C07260=1101.368,312.708,418.200,179.200,17.140,151.820
C07261=1101.362,312.461,418.231,179.196,17.137,151.821
C07262=1101.356,312.212,418.263,179.193,17.135,151.821
C07263=1101.350,311.965,418.294,179.189,17.133,151.821
C07264=1101.345,311.716,418.325,179.186,17.131,151.821
C07265=1101.339,311.469,418.356,179.183,17.129,151.821
C07266=1101.333,311.221,418.387,179.179,17.128,151.822
C07267=1101.327,310.972,418.419,179.175,17.126,151.822
C07268=1101.322,310.725,418.450,179.172,17.124,151.822
C07269=1101.316,310.477,418.481,179.169,17.121,151.822
C07270=1101.310,310.229,418.512,179.165,17.119,151.822
C07271=1101.304,309.981,418.544,179.162,17.117,151.823
C07272=1101.299,309.733,418.575,179.158,17.115,151.823
C07273=1101.293,309.485,418.606,179.156,17.114,151.823
C07274=1101.288,309.237,418.637,179.152,17.112,151.823
C07275=1101.282,308.989,418.667,179.149,17.110,151.824
C07276=1101.276,308.741,418.699,179.145,17.108,151.824
C07277=1101.270,308.493,418.730,179.142,17.106,151.824
C07278=1101.265,308.245,418.761,179.138,17.104,151.824
C07279=1101.259,307.998,418.792,179.135,17.102,151.824
C07280=1101.253,307.749,418.823,179.131,17.100,151.825
C07281=1101.247,307.501,418.853,179.128,17.098,151.825
C07282=1101.242,307.254,418.885,179.124,17.096,151.825
C07283=1101.236,307.006,418.915,179.121,17.094,151.825
C07284=1101.230,306.757,418.947,179.118,17.093,151.826
C07285=1101.225,306.509,418.977,179.115,17.091,151.826
C07286=1101.219,306.262,419.009,179.111,17.089,151.826
C07287=1101.213,306.014,419.039,179.108,17.087,151.826
C07288=1101.208,305.766,419.070,179.104,17.085,151.826
C07289=1101.202,305.517,419.101,179.101,17.083,151.827
C07290=1101.197,305.269,419.132,179.097,17.081,151.827
C07291=1101.191,305.022,419.163,179.094,17.079,151.827
C07292=1101.186,304.774,419.194,179.090,17.078,151.827
C07293=1101.180,304.526,419.224,179.087,17.075,151.828
C07294=1101.174,304.277,419.255,179.084,17.074,151.828
C07295=1101.168,304.029,419.286,179.081,17.072,151.828
C07296=1101.162,303.781,419.316,179.077,17.070,151.828
C07297=1101.154,303.400,419.364,179.072,17.068,151.829
C07298=1101.146,303.018,419.411,179.067,17.065,151.829
C07299=1101.137,302.637,419.458,179.061,17.062,151.830
C07300=1101.128,302.254,419.505,179.056,17.059,151.830
C07301=1101.123,302.006,419.536,179.053,17.057,151.830
C07302=1101.117,301.758,419.567,179.049,17.055,151.830
C07303=1101.111,301.511,419.597,179.045,17.053,151.831
C07304=1101.106,301.262,419.627,179.042,17.051,151.831
C07305=1101.100,301.014,419.658,179.039,17.050,151.831
C07306=1101.095,300.766,419.688,179.036,17.048,151.831
C07307=1101.089,300.518,419.719,179.032,17.046,151.832
C07308=1101.084,300.270,419.749,179.029,17.044,151.832
C07309=1101.078,300.022,419.779,179.025,17.042,151.832
C07310=1101.073,299.774,419.810,179.022,17.040,151.832
C07311=1101.067,299.527,419.841,179.019,17.039,151.833
C07312=1101.061,299.278,419.870,179.015,17.037,151.833
C07313=1101.056,299.030,419.901,179.012,17.035,151.833
C07314=1101.051,298.782,419.932,179.008,17.034,151.834
C07315=1101.045,298.534,419.962,179.005,17.032,151.834
C07316=1101.039,298.286,419.992,179.001,17.030,151.834
C07317=1101.034,298.038,420.023,178.998,17.028,151.834
C07318=1101.028,297.790,420.053,178.995,17.027,151.835
C07319=1101.022,297.542,420.083,178.991,17.025,151.835
C07320=1101.017,297.294,420.114,178.988,17.023,151.835
C07321=1101.011,297.046,420.143,178.984,17.021,151.835
C07322=1101.005,296.798,420.174,178.981,17.019,151.836
C07323=1101.000,296.550,420.204,178.978,17.018,151.836
C07324=1100.994,296.302,420.234,178.974,17.016,151.836
C07325=1100.986,295.953,420.277,178.969,17.014,151.837
C07326=1100.978,295.604,420.319,178.964,17.012,151.837
C07327=1100.970,295.257,420.361,178.960,17.010,151.838
C07328=1100.961,294.908,420.404,178.954,17.007,151.838
C07329=1100.956,294.659,420.433,178.952,17.006,151.838
C07330=1100.950,294.412,420.464,178.948,17.004,151.839
C07331=1100.945,294.164,420.493,178.944,17.002,151.839
C07332=1100.939,293.916,420.523,178.941,17.000,151.839
C07333=1100.934,293.668,420.553,178.938,16.999,151.840
C07334=1100.928,293.420,420.583,178.934,16.997,151.840
C07335=1100.922,293.171,420.613,178.931,16.996,151.840
C07336=1100.917,292.924,420.643,178.927,16.994,151.841
C07337=1100.911,292.675,420.673,178.924,16.992,151.841
C07338=1100.905,292.427,420.703,178.921,16.991,151.841
C07339=1100.900,292.179,420.733,178.917,16.989,151.841
C07340=1100.894,291.931,420.763,178.914,16.987,151.842
C07341=1100.888,291.683,420.793,178.910,16.986,151.842
C07342=1100.883,291.434,420.822,178.907,16.985,151.842
C07343=1100.877,291.186,420.853,178.903,16.983,151.843
C07344=1100.872,290.938,420.882,178.900,16.981,151.843
C07345=1100.866,290.689,420.912,178.896,16.979,151.843
C07346=1100.860,290.442,420.942,178.893,16.978,151.844
C07347=1100.855,290.194,420.971,178.889,16.977,151.844
C07348=1100.849,289.946,421.001,178.886,16.975,151.844
C07349=1100.843,289.678,421.033,178.882,16.973,151.845
C07350=1100.837,289.410,421.065,178.879,16.972,151.845
C07351=1100.830,289.143,421.097,178.875,16.970,151.845
C07352=1100.824,288.875,421.129,178.871,16.968,151.846
C07353=1100.819,288.627,421.159,178.867,16.967,151.846
C07354=1100.814,288.379,421.188,178.864,16.965,151.846
C07355=1100.807,288.132,421.218,178.861,16.964,151.847
C07356=1100.802,287.883,421.248,178.857,16.963,151.847
C07357=1100.796,287.635,421.277,178.853,16.961,151.847
C07358=1100.790,287.387,421.306,178.851,16.960,151.848
C07359=1100.784,287.138,421.336,178.847,16.958,151.848
C07360=1100.779,286.890,421.366,178.843,16.957,151.849
C07361=1100.773,286.642,421.396,178.840,16.955,151.849
C07362=1100.767,286.394,421.425,178.837,16.954,151.849
C07363=1100.762,286.146,421.454,178.833,16.952,151.849
C07364=1100.756,285.898,421.484,178.829,16.950,151.850
C07365=1100.750,285.649,421.513,178.826,16.949,151.850
C07366=1100.745,285.401,421.543,178.823,16.948,151.851
C07367=1100.740,285.153,421.572,178.819,16.946,151.851
C07368=1100.733,284.905,421.601,178.815,16.945,151.851
C07369=1100.728,284.657,421.630,178.812,16.944,151.852
C07370=1100.722,284.408,421.660,178.809,16.942,151.852
C07371=1100.716,284.160,421.689,178.805,16.940,151.852
C07372=1100.711,283.912,421.718,178.801,16.939,151.853
C07373=1100.706,283.664,421.748,178.798,16.938,151.853
C07374=1100.699,283.416,421.777,178.795,16.936,151.853
C07375=1100.694,283.167,421.807,178.791,16.934,151.854
C07376=1100.688,282.920,421.835,178.788,16.933,151.854
C07377=1100.683,282.671,421.865,178.785,16.931,151.854
C07378=1100.678,282.422,421.894,178.781,16.930,151.855
C07379=1100.671,282.174,421.923,178.778,16.929,151.855
C07380=1100.666,281.927,421.952,178.774,16.927,151.856
C07381=1100.660,281.678,421.981,178.771,16.926,151.856
C07382=1100.655,281.430,422.011,178.768,16.925,151.856
C07383=1100.649,281.182,422.041,178.764,16.923,151.857
C07384=1100.644,280.933,422.069,178.760,16.921,151.857
C07385=1100.638,280.685,422.098,178.756,16.920,151.857
C07386=1100.632,280.437,422.127,178.754,16.919,151.858
C07387=1100.626,280.189,422.156,178.750,16.917,151.858
C07388=1100.621,279.941,422.185,178.746,16.916,151.859
C07389=1100.615,279.692,422.214,178.743,16.915,151.859
C07390=1100.609,279.444,422.243,178.739,16.913,151.859
C07391=1100.604,279.196,422.272,178.735,16.912,151.860
C07392=1100.599,278.947,422.301,178.733,16.911,151.860
C07393=1100.592,278.699,422.330,178.729,16.909,151.860
C07394=1100.587,278.452,422.359,178.725,16.908,151.861
C07395=1100.582,278.203,422.388,178.722,16.907,151.861
C07396=1100.575,277.955,422.417,178.718,16.905,151.862
C07397=1100.570,277.707,422.446,178.715,16.903,151.862
C07398=1100.564,277.458,422.474,178.712,16.902,151.862
C07399=1100.558,277.210,422.503,178.708,16.901,151.863
C07400=1100.554,276.962,422.532,178.704,16.900,151.863
C07401=1100.545,276.603,422.574,178.699,16.898,151.864
C07402=1100.537,276.244,422.616,178.695,16.896,151.864
C07403=1100.528,275.886,422.656,178.690,16.894,151.865
C07404=1100.520,275.528,422.698,178.684,16.892,151.865
C07405=1100.515,275.279,422.727,178.681,16.891,151.866
C07406=1100.509,275.031,422.756,178.677,16.890,151.866
C07407=1100.504,274.783,422.784,178.674,16.889,151.867
C07408=1100.498,274.534,422.813,178.671,16.887,151.867
C07409=1100.493,274.287,422.842,178.667,16.886,151.867
C07410=1100.487,274.038,422.870,178.664,16.885,151.868
C07411=1100.481,273.790,422.899,178.660,16.883,151.868
C07412=1100.475,273.542,422.927,178.656,16.882,151.869
C07413=1100.470,273.293,422.956,178.653,16.881,151.869
C07414=1100.464,273.045,422.985,178.650,16.879,151.869
C07415=1100.458,272.796,423.013,178.646,16.878,151.870
C07416=1100.452,272.548,423.042,178.643,16.877,151.870
C07417=1100.447,272.300,423.070,178.639,16.875,151.871
C07418=1100.441,272.052,423.098,178.636,16.875,151.871
C07419=1100.436,271.804,423.128,178.632,16.873,151.871
C07420=1100.430,271.555,423.156,178.628,16.872,151.872
C07421=1100.425,271.307,423.184,178.625,16.871,151.872
C07422=1100.419,271.058,423.212,178.622,16.869,151.873
C07423=1100.412,270.810,423.241,178.619,16.868,151.873
C07424=1100.407,270.562,423.269,178.615,16.867,151.874
C07425=1100.401,270.313,423.298,178.611,16.865,151.874
C07426=1100.397,270.065,423.326,178.608,16.864,151.874
C07427=1100.391,269.816,423.355,178.604,16.863,151.875
C07428=1100.385,269.569,423.383,178.601,16.862,151.875
C07429=1100.379,269.320,423.412,178.598,16.861,151.876
C07430=1100.374,269.072,423.439,178.594,16.860,151.876
C07431=1100.368,268.823,423.468,178.591,16.859,151.876
C07432=1100.362,268.575,423.496,178.587,16.857,151.877
C07433=1100.356,268.326,423.524,178.584,16.856,151.877
C07434=1100.351,268.078,423.552,178.580,16.855,151.878
C07435=1100.345,267.830,423.580,178.576,16.853,151.878
C07436=1100.340,267.582,423.609,178.573,16.853,151.879
C07437=1100.334,267.333,423.637,178.569,16.851,151.879
C07438=1100.328,267.085,423.665,178.566,16.850,151.879
C07439=1100.322,266.837,423.694,178.562,16.849,151.880
C07440=1100.317,266.589,423.722,178.559,16.847,151.880
C07441=1100.312,266.341,423.750,178.556,16.846,151.881
C07442=1100.306,266.092,423.778,178.552,16.845,151.881
C07443=1100.300,265.844,423.806,178.549,16.844,151.882
C07444=1100.294,265.595,423.834,178.545,16.843,151.882
C07445=1100.289,265.347,423.862,178.542,16.842,151.882
C07446=1100.283,265.098,423.890,178.538,16.840,151.883
C07447=1100.277,264.850,423.917,178.534,16.839,151.883
C07448=1100.272,264.602,423.945,178.531,16.838,151.884
C07449=1100.266,264.353,423.973,178.528,16.837,151.884
C07450=1100.261,264.105,424.001,178.524,16.836,151.885
C07451=1100.255,263.856,424.030,178.521,16.835,151.885
C07452=1100.249,263.608,424.058,178.517,16.834,151.886
C07453=1100.240,263.253,424.097,178.513,16.832,151.886
C07454=1100.232,262.897,424.137,178.507,16.830,151.887
C07455=1100.224,262.540,424.177,178.502,16.829,151.888
C07456=1100.216,262.185,424.216,178.497,16.827,151.888
C07457=1100.210,261.936,424.245,178.494,16.827,151.889
C07458=1100.205,261.688,424.273,178.490,16.825,151.889
C07459=1100.198,261.439,424.300,178.487,16.825,151.890
C07460=1100.193,261.191,424.328,178.483,16.823,151.890
C07461=1100.188,260.943,424.356,178.480,16.822,151.890
C07462=1100.181,260.695,424.383,178.476,16.821,151.891
C07463=1100.176,260.446,424.411,178.473,16.820,151.891
C07464=1100.171,260.198,424.439,178.469,16.819,151.892
C07465=1100.164,259.950,424.466,178.465,16.818,151.892
C07466=1100.159,259.701,424.494,178.462,16.817,151.893
C07467=1100.153,259.452,424.522,178.458,16.815,151.893
C07468=1100.147,259.205,424.549,178.455,16.815,151.894
C07469=1100.142,258.956,424.576,178.451,16.813,151.894
C07470=1100.136,258.707,424.605,178.448,16.813,151.895
C07471=1100.130,258.459,424.631,178.444,16.811,151.895
C07472=1100.125,258.211,424.659,178.441,16.811,151.896
C07473=1100.118,257.962,424.687,178.437,16.809,151.896
C07474=1100.113,257.714,424.714,178.434,16.809,151.896
C07475=1100.108,257.466,424.742,178.430,16.807,151.897
C07476=1100.102,257.217,424.769,178.427,16.806,151.897
C07477=1100.096,256.968,424.797,178.423,16.805,151.898
C07478=1100.090,256.720,424.824,178.420,16.804,151.898
C07479=1100.085,256.472,424.852,178.416,16.803,151.899
C07480=1100.079,256.223,424.880,178.413,16.802,151.899
C07481=1100.073,255.975,424.907,178.409,16.801,151.900
C07482=1100.068,255.726,424.934,178.406,16.800,151.900
C07483=1100.062,255.478,424.961,178.402,16.799,151.901
C07484=1100.056,255.229,424.989,178.399,16.798,151.901
C07485=1100.051,254.981,425.016,178.395,16.797,151.902
C07486=1100.045,254.733,425.044,178.392,16.796,151.902
C07487=1100.039,254.484,425.070,178.388,16.795,151.902
C07488=1100.034,254.235,425.098,178.385,16.794,151.903
C07489=1100.028,253.987,425.125,178.381,16.793,151.903
C07490=1100.023,253.739,425.153,178.378,16.792,151.904
C07491=1100.017,253.490,425.179,178.375,16.791,151.904
C07492=1100.012,253.242,425.207,178.371,16.790,151.905
C07493=1100.006,252.994,425.234,178.368,16.788,151.905
C07494=1100.000,252.744,425.261,178.364,16.788,151.906
C07495=1099.994,252.496,425.288,178.360,16.787,151.906
C07496=1099.989,252.248,425.316,178.357,16.786,151.907
C07497=1099.983,252.000,425.343,178.353,16.785,151.907
C07498=1099.978,251.751,425.370,178.350,16.784,151.908
C07499=1099.973,251.503,425.397,178.346,16.783,151.908
C07500=1099.967,251.253,425.424,178.344,16.782,151.908
C07501=1099.961,251.005,425.452,178.340,16.780,151.909
C07502=1099.956,250.757,425.479,178.337,16.779,151.909
C07503=1099.950,250.508,425.505,178.333,16.778,151.910
C07504=1099.945,250.260,425.533,178.329,16.778,151.910
C07505=1099.937,249.901,425.571,178.325,16.776,151.911
C07506=1099.929,249.543,425.611,178.319,16.775,151.912
C07507=1099.921,249.184,425.649,178.314,16.773,151.913
C07508=1099.913,248.825,425.688,178.310,16.772,151.913
C07509=1099.907,248.577,425.715,178.306,16.771,151.914
C07510=1099.902,248.329,425.742,178.303,16.770,151.914
C07511=1099.896,248.079,425.769,178.299,16.768,151.915
C07512=1099.890,247.831,425.796,178.295,16.768,151.915
C07513=1099.885,247.583,425.822,178.292,16.766,151.915
C07514=1099.879,247.334,425.850,178.288,16.766,151.916
C07515=1099.874,247.086,425.876,178.285,16.764,151.916
C07516=1099.868,246.837,425.903,178.282,16.764,151.917
C07517=1099.862,246.589,425.930,178.278,16.763,151.917
C07518=1099.857,246.340,425.957,178.275,16.762,151.918
C07519=1099.851,246.092,425.984,178.271,16.761,151.918
C07520=1099.846,245.843,426.010,178.267,16.760,151.919
C07521=1099.840,245.595,426.037,178.264,16.759,151.919
C07522=1099.835,245.346,426.064,178.260,16.758,151.920
C07523=1099.829,245.098,426.091,178.257,16.757,151.920
C07524=1099.823,244.850,426.117,178.253,16.756,151.921
C07525=1099.818,244.601,426.143,178.250,16.755,151.921
C07526=1099.812,244.352,426.170,178.246,16.754,151.922
C07527=1099.807,244.104,426.197,178.243,16.753,151.922
C07528=1099.801,243.855,426.224,178.240,16.753,151.923
C07529=1099.795,243.607,426.250,178.236,16.752,151.923
C07530=1099.790,243.358,426.276,178.233,16.751,151.924
C07531=1099.784,243.110,426.303,178.229,16.750,151.924
C07532=1099.778,242.861,426.330,178.226,16.749,151.925
C07533=1099.773,242.613,426.356,178.222,16.747,151.925
C07534=1099.767,242.364,426.382,178.219,16.747,151.926
C07535=1099.761,242.116,426.409,178.216,16.746,151.926
C07536=1099.756,241.867,426.436,178.212,16.745,151.927
C07537=1099.750,241.619,426.462,178.208,16.745,151.927
C07538=1099.744,241.370,426.488,178.205,16.743,151.928
C07539=1099.739,241.122,426.515,178.201,16.743,151.928
C07540=1099.733,240.873,426.541,178.198,16.742,151.929
C07541=1099.727,240.624,426.567,178.194,16.741,151.929
C07542=1099.722,240.376,426.594,178.191,16.740,151.930
C07543=1099.716,240.127,426.620,178.187,16.739,151.930
C07544=1099.710,239.878,426.647,178.184,16.738,151.931
C07545=1099.705,239.630,426.673,178.180,16.737,151.931
C07546=1099.699,239.381,426.699,178.177,16.736,151.932
C07547=1099.693,239.133,426.726,178.174,16.736,151.932
C07548=1099.688,238.884,426.752,178.170,16.735,151.933
C07549=1099.682,238.635,426.778,178.167,16.734,151.933
C07550=1099.677,238.386,426.804,178.163,16.733,151.934
C07551=1099.671,238.138,426.831,178.160,16.732,151.934
C07552=1099.665,237.889,426.857,178.156,16.732,151.935
C07553=1099.660,237.641,426.884,178.152,16.731,151.935
C07554=1099.654,237.392,426.910,178.149,16.730,151.936
C07555=1099.649,237.144,426.936,178.145,16.728,151.936
C07556=1099.643,236.895,426.961,178.142,16.728,151.937
C07557=1099.634,236.529,427.001,178.137,16.727,151.938
C07558=1099.626,236.164,427.039,178.132,16.725,151.938
C07559=1099.618,235.798,427.077,178.127,16.724,151.939
C07560=1099.610,235.433,427.115,178.122,16.723,151.940
C07561=1099.604,235.184,427.141,178.119,16.722,151.940
C07562=1099.598,234.936,427.168,178.115,16.721,151.941
C07563=1099.593,234.688,427.193,178.111,16.721,151.941
C07564=1099.587,234.439,427.219,178.108,16.720,151.942
C07565=1099.582,234.191,427.246,178.104,16.719,151.942
C07566=1099.576,233.942,427.271,178.101,16.718,151.943
C07567=1099.571,233.693,427.297,178.098,16.718,151.943
C07568=1099.564,233.444,427.323,178.094,16.716,151.944
C07569=1099.559,233.196,427.349,178.091,16.716,151.944
C07570=1099.554,232.947,427.375,178.087,16.714,151.945
C07571=1099.548,232.698,427.401,178.084,16.714,151.945
C07572=1099.542,232.450,427.426,178.081,16.713,151.946
C07573=1099.536,232.201,427.453,178.077,16.712,151.946
C07574=1099.532,231.953,427.478,178.074,16.711,151.947
C07575=1099.525,231.704,427.504,178.070,16.711,151.948
C07576=1099.520,231.455,427.530,178.066,16.710,151.948
C07577=1099.514,231.206,427.556,178.063,16.709,151.949
C07578=1099.509,230.959,427.582,178.060,16.708,151.949
C07579=1099.503,230.710,427.607,178.056,16.707,151.950
C07580=1099.498,230.461,427.633,178.053,16.707,151.950
C07581=1099.491,230.212,427.659,178.050,16.706,151.951
C07582=1099.486,229.963,427.684,178.046,16.705,151.951
C07583=1099.481,229.715,427.710,178.042,16.705,151.952
C07584=1099.475,229.467,427.735,178.039,16.704,151.952
C07585=1099.469,229.218,427.761,178.035,16.703,151.953
C07586=1099.463,228.969,427.787,178.032,16.702,151.953
C07587=1099.458,228.721,427.812,178.029,16.702,151.954
C07588=1099.452,228.472,427.838,178.025,16.700,151.954
C07589=1099.447,228.223,427.863,178.022,16.700,151.955
C07590=1099.440,227.974,427.889,178.018,16.699,151.955
C07591=1099.436,227.726,427.914,178.014,16.698,151.956
C07592=1099.429,227.477,427.940,178.011,16.698,151.956
C07593=1099.424,227.228,427.966,178.008,16.697,151.957
C07594=1099.418,226.980,427.991,178.004,16.696,151.957
C07595=1099.413,226.731,428.017,178.001,16.695,151.958
C07596=1099.407,226.483,428.042,177.998,16.695,151.959
C07597=1099.401,226.234,428.068,177.994,16.694,151.959
C07598=1099.395,225.986,428.093,177.991,16.693,151.960
C07599=1099.390,225.737,428.119,177.987,16.693,151.960
C07600=1099.384,225.488,428.144,177.983,16.692,151.961
C07601=1099.379,225.240,428.170,177.980,16.691,151.961
C07602=1099.373,224.991,428.194,177.977,16.690,151.962
C07603=1099.368,224.742,428.220,177.973,16.689,151.962
C07604=1099.362,224.494,428.245,177.970,16.689,151.963
C07605=1099.356,224.245,428.271,177.967,16.688,151.963
C07606=1099.351,223.997,428.296,177.963,16.687,151.964
C07607=1099.346,223.747,428.321,177.960,16.686,151.964
C07608=1099.340,223.498,428.347,177.956,16.686,151.965
C07609=1099.331,223.125,428.384,177.951,16.685,151.966
C07610=1099.323,222.751,428.422,177.946,16.683,151.966
C07611=1099.314,222.377,428.460,177.941,16.682,151.967
C07612=1099.306,222.003,428.498,177.936,16.681,151.968
C07613=1099.300,221.754,428.523,177.932,16.680,151.968
C07614=1099.295,221.506,428.548,177.928,16.679,151.969
C07615=1099.289,221.257,428.574,177.925,16.679,151.970
C07616=1099.283,221.008,428.599,177.922,16.678,151.970
C07617=1099.278,220.760,428.624,177.919,16.678,151.971
C07618=1099.272,220.510,428.649,177.915,16.677,151.971
C07619=1099.266,220.261,428.675,177.911,16.676,151.972
C07620=1099.261,220.014,428.700,177.908,16.676,151.972
C07621=1099.255,219.764,428.724,177.904,16.675,151.973
C07622=1099.249,219.516,428.749,177.901,16.674,151.973
C07623=1099.243,219.267,428.774,177.898,16.674,151.974
C07624=1099.238,219.019,428.799,177.895,16.673,151.975
C07625=1099.232,218.770,428.825,177.890,16.672,151.975
C07626=1099.227,218.521,428.849,177.888,16.671,151.976
C07627=1099.221,218.273,428.874,177.884,16.671,151.976
C07628=1099.215,218.023,428.899,177.880,16.670,151.977
C07629=1099.210,217.775,428.924,177.877,16.669,151.977
C07630=1099.204,217.526,428.949,177.874,16.669,151.978
C07631=1099.198,217.278,428.974,177.871,16.668,151.978
C07632=1099.193,217.029,428.999,177.867,16.667,151.979
C07633=1099.187,216.780,429.023,177.863,16.667,151.979
C07634=1099.182,216.531,429.049,177.860,16.666,151.980
C07635=1099.177,216.282,429.073,177.857,16.666,151.980
C07636=1099.170,216.034,429.098,177.853,16.665,151.981
C07637=1099.165,215.785,429.123,177.850,16.664,151.981
C07638=1099.159,215.536,429.147,177.847,16.663,151.982
C07639=1099.153,215.288,429.172,177.843,16.663,151.983
C07640=1099.148,215.039,429.197,177.839,16.662,151.983
C07641=1099.142,214.790,429.221,177.836,16.661,151.984
C07642=1099.137,214.542,429.247,177.833,16.661,151.984
C07643=1099.132,214.293,429.271,177.830,16.660,151.985
C07644=1099.126,214.044,429.296,177.826,16.659,151.985
C07645=1099.120,213.795,429.321,177.822,16.659,151.986
C07646=1099.115,213.547,429.345,177.819,16.658,151.986
C07647=1099.109,213.298,429.369,177.816,16.657,151.987
C07648=1099.103,213.049,429.395,177.812,16.656,151.987
C07649=1099.098,212.801,429.419,177.809,16.656,151.988
C07650=1099.092,212.552,429.444,177.806,16.655,151.988
C07651=1099.087,212.303,429.468,177.802,16.655,151.989
C07652=1099.081,212.054,429.493,177.798,16.654,151.990
C07653=1099.075,211.806,429.518,177.795,16.653,151.990
C07654=1099.070,211.557,429.542,177.792,16.653,151.991
C07655=1099.064,211.308,429.566,177.789,16.652,151.991
C07656=1099.059,211.059,429.591,177.785,16.651,151.992
C07657=1099.053,210.810,429.615,177.781,16.651,151.992
C07658=1099.047,210.562,429.640,177.778,16.650,151.993
C07659=1099.042,210.313,429.664,177.775,16.650,151.993
C07660=1099.035,210.064,429.689,177.772,16.649,151.994
C07661=1099.028,209.694,429.725,177.767,16.648,151.995
C07662=1099.019,209.324,429.761,177.761,16.647,151.995
C07663=1099.010,208.954,429.798,177.756,16.646,151.996
C07664=1099.002,208.584,429.834,177.751,16.645,151.997
C07665=1098.979,207.575,429.932,177.709,16.631,152.003
C07666=1098.974,207.326,429.956,177.705,16.631,152.003
C07667=1098.968,207.078,429.980,177.702,16.632,152.004
C07668=1098.963,206.829,430.003,177.698,16.632,152.005
C07669=1098.957,206.579,430.028,177.694,16.632,152.006
C07670=1098.951,206.331,430.052,177.691,16.632,152.007
C07671=1098.945,206.082,430.076,177.687,16.632,152.007
C07672=1098.940,205.834,430.100,177.683,16.632,152.008
C07673=1098.934,205.585,430.124,177.680,16.632,152.009
C07674=1098.928,205.336,430.147,177.676,16.633,152.010
C07675=1098.923,205.087,430.172,177.673,16.633,152.010
C07676=1098.918,204.839,430.196,177.670,16.633,152.011
C07677=1098.911,204.590,430.220,177.666,16.634,152.012
C07678=1098.906,204.340,430.244,177.662,16.634,152.013
C07679=1098.901,204.092,430.268,177.658,16.634,152.014
C07680=1098.895,203.843,430.291,177.655,16.634,152.014
C07681=1098.890,203.594,430.315,177.651,16.634,152.015
C07682=1098.883,203.345,430.339,177.648,16.635,152.016
C07683=1098.878,203.097,430.363,177.644,16.635,152.017
C07684=1098.873,202.848,430.387,177.640,16.635,152.017
C07685=1098.867,202.599,430.410,177.637,16.635,152.018
C07686=1098.862,202.351,430.435,177.633,16.635,152.019
C07687=1098.855,202.101,430.458,177.630,16.636,152.020
C07688=1098.850,201.852,430.482,177.627,16.636,152.020
C07689=1098.844,201.604,430.506,177.623,16.636,152.021
C07690=1098.838,201.355,430.529,177.619,16.637,152.022
C07691=1098.832,201.106,430.554,177.616,16.637,152.023
C07692=1098.826,200.858,430.577,177.612,16.637,152.024
C07693=1098.821,200.609,430.601,177.608,16.637,152.024
C07694=1098.815,200.360,430.624,177.605,16.637,152.025
C07695=1098.810,200.111,430.648,177.601,16.638,152.026
C07696=1098.804,199.862,430.672,177.598,16.638,152.027
C07697=1098.798,199.613,430.695,177.594,16.639,152.027
C07698=1098.793,199.365,430.719,177.591,16.639,152.028
C07699=1098.787,199.116,430.742,177.587,16.639,152.029
C07700=1098.781,198.867,430.766,177.583,16.639,152.030
C07701=1098.776,198.618,430.789,177.580,16.639,152.030
C07702=1098.769,198.369,430.813,177.576,16.639,152.031
C07703=1098.764,198.120,430.837,177.573,16.639,152.032
C07704=1098.758,197.872,430.861,177.569,16.639,152.033
C07705=1098.752,197.623,430.883,177.566,16.640,152.033
C07706=1098.747,197.374,430.908,177.562,16.641,152.034
C07707=1098.741,197.125,430.931,177.559,16.641,152.035
C07708=1098.736,196.876,430.954,177.555,16.641,152.036
C07709=1098.730,196.628,430.978,177.552,16.641,152.036
C07710=1098.725,196.379,431.001,177.548,16.641,152.037
C07711=1098.718,196.129,431.024,177.544,16.641,152.038
C07712=1098.713,195.881,431.048,177.541,16.641,152.039
C07713=1098.707,195.632,431.071,177.537,16.641,152.039
C07714=1098.701,195.383,431.094,177.534,16.642,152.040
C07715=1098.696,195.134,431.119,177.531,16.642,152.041
C07716=1098.690,194.885,431.141,177.527,16.642,152.042
C07717=1098.685,194.637,431.164,177.524,16.642,152.042
C07718=1098.679,194.388,431.188,177.520,16.643,152.043
C07719=1098.674,194.139,431.212,177.516,16.643,152.044
C07720=1098.668,193.890,431.235,177.513,16.643,152.045
C07721=1098.662,193.641,431.258,177.509,16.643,152.045
C07722=1098.657,193.393,431.282,177.507,16.643,152.046
C07723=1098.651,193.144,431.305,177.503,16.643,152.047
C07724=1098.645,192.895,431.328,177.499,16.644,152.048
C07725=1098.640,192.646,431.351,177.496,16.644,152.048
C07726=1098.633,192.373,431.377,177.492,16.644,152.049
C07727=1098.627,192.099,431.402,177.488,16.644,152.050
C07728=1098.621,191.825,431.428,177.485,16.644,152.051
C07729=1098.615,191.552,431.453,177.480,16.644,152.052
C07730=1098.610,191.303,431.476,177.477,16.645,152.052
C07731=1098.604,191.054,431.499,177.474,16.645,152.053
C07732=1098.599,190.805,431.522,177.470,16.645,152.054
C07733=1098.593,190.557,431.546,177.467,16.645,152.054
C07734=1098.588,190.307,431.569,177.463,16.645,152.055
C07735=1098.582,190.058,431.592,177.460,16.645,152.056
C07736=1098.576,189.810,431.615,177.456,16.645,152.057
C07737=1098.570,189.561,431.638,177.452,16.645,152.058
C07738=1098.565,189.312,431.661,177.450,16.646,152.058
C07739=1098.560,189.063,431.685,177.446,16.646,152.059
C07740=1098.554,188.814,431.708,177.442,16.646,152.060
C07741=1098.548,188.565,431.731,177.439,16.646,152.060
C07742=1098.543,188.316,431.753,177.435,16.646,152.061
C07743=1098.537,188.068,431.776,177.432,16.646,152.062
C07744=1098.532,187.819,431.799,177.428,16.646,152.062
C07745=1098.526,187.570,431.822,177.426,16.646,152.063
C07746=1098.521,187.321,431.845,177.422,16.646,152.064
C07747=1098.515,187.072,431.868,177.418,16.646,152.065
C07748=1098.509,186.823,431.891,177.415,16.647,152.065
C07749=1098.504,186.574,431.914,177.411,16.647,152.066
C07750=1098.498,186.325,431.937,177.408,16.647,152.067
C07751=1098.493,186.076,431.959,177.405,16.647,152.067
C07752=1098.487,185.827,431.982,177.402,16.647,152.068
C07753=1098.482,185.578,432.006,177.398,16.647,152.069
C07754=1098.477,185.329,432.029,177.395,16.647,152.069
C07755=1098.471,185.080,432.052,177.391,16.647,152.070
C07756=1098.465,184.832,432.074,177.388,16.647,152.071
C07757=1098.459,184.583,432.097,177.384,16.647,152.072
C07758=1098.453,184.333,432.119,177.381,16.648,152.072
C07759=1098.448,184.084,432.142,177.378,16.648,152.073
C07760=1098.443,183.836,432.165,177.374,16.648,152.074
C07761=1098.437,183.587,432.188,177.370,16.648,152.075
C07762=1098.430,183.339,432.210,177.367,16.648,152.075
C07763=1098.425,183.090,432.233,177.364,16.649,152.076
C07764=1098.419,182.840,432.255,177.361,16.649,152.077
C07765=1098.413,182.591,432.278,177.357,16.649,152.077
C07766=1098.408,182.343,432.301,177.354,16.649,152.078
C07767=1098.401,182.094,432.323,177.350,16.649,152.079
C07768=1098.396,181.844,432.346,177.346,16.649,152.080
C07769=1098.390,181.596,432.368,177.344,16.649,152.080
C07770=1098.385,181.347,432.391,177.340,16.649,152.081
C07771=1098.379,181.098,432.413,177.337,16.649,152.082
C07772=1098.373,180.849,432.436,177.333,16.650,152.082
C07773=1098.367,180.600,432.459,177.330,16.650,152.083
C07774=1098.362,180.351,432.481,177.327,16.650,152.084
C07775=1098.355,180.102,432.503,177.323,16.650,152.085
C07776=1098.350,179.853,432.526,177.320,16.650,152.085
C07777=1098.345,179.605,432.548,177.316,16.650,152.086
C07778=1098.339,179.356,432.571,177.313,16.650,152.087
C07779=1098.333,179.107,432.593,177.309,16.650,152.087
C07780=1098.327,178.858,432.615,177.306,16.651,152.088
C07781=1098.322,178.609,432.638,177.303,16.651,152.089
C07782=1098.317,178.360,432.660,177.299,16.651,152.090
C07783=1098.310,178.111,432.683,177.296,16.651,152.090
C07784=1098.305,177.862,432.705,177.292,16.651,152.091
C07785=1098.299,177.613,432.728,177.290,16.651,152.092
C07786=1098.293,177.364,432.749,177.286,16.651,152.092
C07787=1098.288,177.115,432.772,177.283,16.651,152.093
C07788=1098.282,176.866,432.794,177.279,16.651,152.094
C07789=1098.276,176.617,432.817,177.276,16.651,152.094
C07790=1098.270,176.343,432.841,177.272,16.651,152.095
C07791=1098.264,176.070,432.865,177.268,16.651,152.096
C07792=1098.258,175.795,432.890,177.265,16.652,152.097
C07793=1098.251,175.521,432.915,177.261,16.652,152.098
C07794=1098.246,175.272,432.937,177.258,16.652,152.098
C07795=1098.240,175.024,432.959,177.254,16.652,152.099
C07796=1098.234,174.774,432.981,177.252,16.652,152.100
C07797=1098.229,174.525,433.004,177.248,16.652,152.100
C07798=1098.224,174.277,433.026,177.244,16.652,152.101
C07799=1098.218,174.027,433.048,177.241,16.652,152.102
C07800=1098.212,173.779,433.070,177.238,16.652,152.102
C07801=1098.206,173.530,433.092,177.235,16.653,152.103
C07802=1098.201,173.281,433.114,177.231,16.653,152.104
C07803=1098.195,173.032,433.137,177.228,16.652,152.104
C07804=1098.190,172.783,433.158,177.225,16.652,152.105
C07805=1098.184,172.534,433.180,177.221,16.652,152.106
C07806=1098.178,172.285,433.203,177.219,16.653,152.106
C07807=1098.173,172.036,433.225,177.215,16.653,152.107
C07808=1098.167,171.787,433.247,177.211,16.653,152.108
C07809=1098.161,171.538,433.269,177.208,16.653,152.108
C07810=1098.156,171.289,433.291,177.205,16.653,152.109
C07811=1098.150,171.040,433.313,177.202,16.653,152.110
C07812=1098.145,170.791,433.335,177.198,16.653,152.110
C07813=1098.139,170.542,433.356,177.195,16.653,152.111
C07814=1098.133,170.293,433.379,177.192,16.653,152.112
C07815=1098.128,170.045,433.400,177.189,16.653,152.112
C07816=1098.122,169.795,433.423,177.186,16.653,152.113
C07817=1098.117,169.546,433.445,177.182,16.653,152.114
C07818=1098.111,169.297,433.466,177.179,16.652,152.114
C07819=1098.106,169.048,433.489,177.175,16.653,152.115
C07820=1098.100,168.800,433.510,177.173,16.653,152.115
C07821=1098.095,168.550,433.533,177.169,16.653,152.116
C07822=1098.089,168.302,433.554,177.166,16.653,152.117
C07823=1098.084,168.052,433.576,177.162,16.652,152.117
C07824=1098.078,167.804,433.597,177.160,16.653,152.118
C07825=1098.073,167.554,433.620,177.156,16.653,152.119
C07826=1098.067,167.306,433.641,177.153,16.653,152.119
C07827=1098.062,167.056,433.663,177.150,16.652,152.120
C07828=1098.055,166.807,433.685,177.146,16.652,152.121
C07829=1098.051,166.558,433.707,177.144,16.653,152.121
C07830=1098.044,166.309,433.728,177.140,16.653,152.122
C07831=1098.040,166.060,433.750,177.137,16.652,152.123
C07832=1098.033,165.811,433.772,177.133,16.652,152.123
C07833=1098.028,165.562,433.793,177.131,16.652,152.124
C07834=1098.022,165.313,433.815,177.127,16.652,152.125
C07835=1098.017,165.064,433.837,177.124,16.652,152.125
C07836=1098.012,164.816,433.858,177.120,16.652,152.126
C07837=1098.006,164.566,433.880,177.117,16.652,152.126
C07838=1098.001,164.318,433.902,177.115,16.652,152.127
C07839=1097.995,164.068,433.924,177.111,16.652,152.128
C07840=1097.990,163.820,433.945,177.108,16.652,152.128
C07841=1097.984,163.570,433.967,177.104,16.652,152.129
C07842=1097.978,163.322,433.988,177.102,16.652,152.130
C07843=1097.973,163.072,434.011,177.099,16.651,152.130
C07844=1097.967,162.824,434.032,177.095,16.651,152.131
C07845=1097.963,162.575,434.054,177.092,16.651,152.131
C07846=1097.957,162.325,434.075,177.088,16.651,152.132
C07847=1097.951,162.077,434.096,177.086,16.651,152.133
C07848=1097.946,161.827,434.118,177.083,16.651,152.133
C07849=1097.940,161.579,434.139,177.079,16.651,152.134
C07850=1097.934,161.329,434.161,177.076,16.651,152.135
C07851=1097.929,161.081,434.183,177.073,16.651,152.135
C07852=1097.923,160.831,434.204,177.070,16.651,152.136
C07853=1097.918,160.582,434.225,177.067,16.650,152.136
C07854=1097.911,160.308,434.249,177.063,16.651,152.137
C07855=1097.905,160.034,434.272,177.059,16.651,152.138
C07856=1097.899,159.759,434.296,177.056,16.651,152.139
C07857=1097.892,159.485,434.320,177.052,16.651,152.139
C07858=1097.887,159.236,434.340,177.049,16.650,152.140
C07859=1097.881,158.987,434.362,177.047,16.651,152.140
C07860=1097.875,158.738,434.383,177.043,16.651,152.141
C07861=1097.871,158.489,434.404,177.040,16.650,152.142
C07862=1097.865,158.239,434.426,177.036,16.650,152.142
C07863=1097.859,157.991,434.447,177.034,16.650,152.143
C07864=1097.853,157.741,434.468,177.031,16.650,152.144
C07865=1097.848,157.493,434.489,177.027,16.650,152.144
C07866=1097.842,157.244,434.511,177.024,16.650,152.145
C07867=1097.836,156.994,434.532,177.021,16.650,152.145
C07868=1097.831,156.746,434.553,177.018,16.650,152.146
C07869=1097.825,156.496,434.575,177.015,16.650,152.147
C07870=1097.820,156.247,434.596,177.011,16.649,152.147
C07871=1097.814,155.999,434.617,177.009,16.649,152.148
C07872=1097.809,155.749,434.638,177.005,16.649,152.148
C07873=1097.803,155.500,434.659,177.002,16.649,152.149
C07874=1097.797,155.251,434.681,176.999,16.649,152.150
C07875=1097.792,155.002,434.701,176.996,16.649,152.150
C07876=1097.786,154.753,434.723,176.993,16.649,152.151
C07877=1097.780,154.504,434.743,176.989,16.649,152.151
C07878=1097.775,154.255,434.765,176.987,16.649,152.152
C07879=1097.769,154.006,434.785,176.983,16.649,152.153
C07880=1097.763,153.757,434.807,176.980,16.648,152.153
C07881=1097.758,153.508,434.827,176.977,16.648,152.154
C07882=1097.752,153.259,434.849,176.974,16.649,152.155
C07883=1097.747,153.009,434.870,176.971,16.648,152.155
C07884=1097.741,152.761,434.891,176.968,16.648,152.156
C07885=1097.736,152.512,434.912,176.964,16.648,152.156
C07886=1097.730,152.263,434.933,176.962,16.648,152.157
C07887=1097.724,152.013,434.954,176.958,16.648,152.158
C07888=1097.719,151.764,434.974,176.955,16.647,152.158
C07889=1097.712,151.515,434.995,176.953,16.648,152.159
C07890=1097.707,151.266,435.016,176.949,16.647,152.159
C07891=1097.701,151.018,435.037,176.946,16.647,152.160
C07892=1097.696,150.769,435.058,176.943,16.647,152.160
C07893=1097.690,150.519,435.079,176.940,16.647,152.161
C07894=1097.685,150.270,435.100,176.937,16.647,152.162
C07895=1097.679,150.021,435.120,176.934,16.646,152.162
C07896=1097.674,149.771,435.141,176.931,16.647,152.163
C07897=1097.668,149.523,435.163,176.928,16.646,152.163
C07898=1097.663,149.274,435.183,176.925,16.646,152.164
C07899=1097.657,149.025,435.203,176.921,16.645,152.165
C07900=1097.651,148.776,435.225,176.919,16.646,152.165
C07901=1097.645,148.527,435.245,176.915,16.646,152.166
C07902=1097.640,148.277,435.266,176.912,16.645,152.166
C07903=1097.635,148.029,435.287,176.910,16.646,152.167
C07904=1097.628,147.779,435.307,176.906,16.645,152.167
C07905=1097.623,147.530,435.328,176.903,16.645,152.168
C07906=1097.617,147.281,435.349,176.900,16.644,152.169
C07907=1097.612,147.033,435.370,176.897,16.645,152.169
C07908=1097.605,146.783,435.390,176.894,16.644,152.170
C07909=1097.600,146.534,435.411,176.891,16.644,152.170
C07910=1097.595,146.285,435.431,176.888,16.645,152.171
C07911=1097.589,146.036,435.452,176.885,16.644,152.172
C07912=1097.583,145.787,435.473,176.882,16.644,152.172
C07913=1097.577,145.538,435.493,176.878,16.643,152.173
C07914=1097.572,145.289,435.514,176.876,16.644,152.173
C07915=1097.567,145.040,435.535,176.873,16.643,152.174
C07916=1097.561,144.791,435.554,176.869,16.643,152.174
C07917=1097.555,144.541,435.575,176.867,16.643,152.175
C07918=1097.549,144.267,435.598,176.864,16.643,152.176
C07919=1097.542,143.992,435.621,176.860,16.643,152.176
C07920=1097.537,143.718,435.644,176.857,16.642,152.177
C07921=1097.530,143.442,435.666,176.854,16.642,152.177
C07922=1097.525,143.193,435.686,176.850,16.642,152.178
C07923=1097.519,142.944,435.707,176.847,16.641,152.179
C07924=1097.513,142.695,435.727,176.845,16.642,152.179
C07925=1097.508,142.446,435.747,176.841,16.641,152.180
C07926=1097.503,142.197,435.768,176.838,16.641,152.180
C07927=1097.497,141.949,435.789,176.836,16.641,152.181
C07928=1097.491,141.699,435.809,176.832,16.641,152.181
C07929=1097.485,141.450,435.830,176.829,16.640,152.182
C07930=1097.480,141.200,435.849,176.827,16.640,152.183
C07931=1097.474,140.951,435.870,176.824,16.640,152.183
C07932=1097.469,140.703,435.890,176.820,16.639,152.184
C07933=1097.463,140.453,435.910,176.817,16.639,152.184
C07934=1097.458,140.204,435.931,176.815,16.639,152.185
C07935=1097.452,139.955,435.951,176.811,16.639,152.185
C07936=1097.446,139.706,435.972,176.808,16.638,152.186
C07937=1097.440,139.457,435.992,176.806,16.639,152.186
C07938=1097.435,139.208,436.012,176.802,16.638,152.187
C07939=1097.429,138.959,436.032,176.799,16.638,152.187
C07940=1097.424,138.710,436.053,176.797,16.638,152.188
C07941=1097.418,138.461,436.073,176.794,16.637,152.188
C07942=1097.412,138.212,436.093,176.790,16.637,152.189
C07943=1097.407,137.962,436.113,176.788,16.637,152.190
C07944=1097.401,137.713,436.133,176.785,16.637,152.190
C07945=1097.395,137.464,436.153,176.781,16.636,152.191
C07946=1097.390,137.215,436.174,176.779,16.637,152.191
C07947=1097.384,136.966,436.194,176.776,16.636,152.192
C07948=1097.378,136.717,436.214,176.773,16.635,152.192
C07949=1097.373,136.467,436.234,176.770,16.636,152.193
C07950=1097.367,136.218,436.254,176.767,16.635,152.193
C07951=1097.361,135.969,436.274,176.764,16.635,152.194
C07952=1097.355,135.721,436.294,176.762,16.635,152.194
C07953=1097.350,135.471,436.314,176.758,16.634,152.195
C07954=1097.344,135.222,436.334,176.755,16.634,152.196
C07955=1097.339,134.973,436.355,176.753,16.634,152.196
C07956=1097.333,134.724,436.374,176.750,16.633,152.196
C07957=1097.328,134.474,436.394,176.746,16.633,152.197
C07958=1097.322,134.225,436.414,176.744,16.633,152.198
C07959=1097.316,133.977,436.434,176.741,16.633,152.198
C07960=1097.311,133.727,436.454,176.738,16.632,152.199
C07961=1097.305,133.478,436.474,176.735,16.632,152.199
C07962=1097.300,133.229,436.495,176.732,16.632,152.200
C07963=1097.294,132.980,436.514,176.729,16.631,152.200
C07964=1097.288,132.731,436.534,176.726,16.631,152.201
C07965=1097.283,132.482,436.554,176.723,16.631,152.201
C07966=1097.277,132.232,436.574,176.720,16.630,152.202
C07967=1097.271,131.983,436.594,176.718,16.630,152.202
C07968=1097.265,131.735,436.614,176.715,16.630,152.203
C07969=1097.261,131.485,436.633,176.711,16.629,152.203
C07970=1097.255,131.236,436.653,176.709,16.629,152.204
C07971=1097.249,130.987,436.673,176.706,16.629,152.204
C07972=1097.243,130.738,436.692,176.703,16.628,152.205
C07973=1097.237,130.488,436.712,176.700,16.629,152.205
C07974=1097.232,130.239,436.732,176.697,16.628,152.206
C07975=1097.226,129.990,436.752,176.694,16.628,152.206
C07976=1097.220,129.741,436.771,176.691,16.628,152.207
C07977=1097.214,129.492,436.791,176.688,16.627,152.207
C07978=1097.209,129.243,436.811,176.685,16.627,152.208
C07979=1097.203,128.994,436.831,176.683,16.627,152.209
C07980=1097.198,128.744,436.850,176.680,16.626,152.209
C07981=1097.192,128.495,436.870,176.676,16.626,152.210
C07982=1097.185,128.221,436.892,176.674,16.626,152.210
C07983=1097.179,127.945,436.914,176.671,16.625,152.211
C07984=1097.173,127.671,436.935,176.667,16.625,152.211
C07985=1097.167,127.396,436.957,176.664,16.625,152.212
C07986=1097.161,127.147,436.976,176.661,16.624,152.212
C07987=1097.155,126.898,436.996,176.658,16.624,152.213
C07988=1097.149,126.649,437.015,176.656,16.623,152.213
C07989=1097.144,126.399,437.035,176.652,16.623,152.214
C07990=1097.138,126.150,437.055,176.650,16.623,152.214
C07991=1097.133,125.901,437.075,176.647,16.622,152.215
C07992=1097.127,125.651,437.094,176.644,16.622,152.215
C07993=1097.121,125.402,437.114,176.642,16.622,152.216
C07994=1097.115,125.153,437.133,176.639,16.621,152.216
C07995=1097.110,124.904,437.152,176.635,16.621,152.217
C07996=1097.104,124.655,437.172,176.633,16.621,152.217
C07997=1097.098,124.406,437.191,176.630,16.620,152.218
C07998=1097.093,124.157,437.210,176.627,16.619,152.218
C07999=1097.087,123.908,437.230,176.624,16.619,152.219
C08000=1097.081,123.658,437.249,176.621,16.619,152.219
C08001=1097.075,123.409,437.269,176.619,16.619,152.220
C08002=1097.071,123.160,437.289,176.616,16.618,152.220
C08003=1097.065,122.911,437.308,176.613,16.618,152.221
C08004=1097.059,122.662,437.327,176.611,16.617,152.221
C08005=1097.054,122.412,437.347,176.607,16.617,152.222
C08006=1097.048,122.163,437.367,176.604,16.616,152.222
C08007=1097.042,121.914,437.386,176.602,16.616,152.223
C08008=1097.037,121.665,437.405,176.599,16.616,152.223
C08009=1097.031,121.416,437.424,176.596,16.615,152.224
C08010=1097.026,121.166,437.443,176.593,16.615,152.224
C08011=1097.020,120.917,437.462,176.591,16.614,152.224
C08012=1097.014,120.668,437.482,176.588,16.614,152.225
C08013=1097.009,120.419,437.501,176.585,16.614,152.225
C08014=1097.003,120.170,437.521,176.582,16.613,152.226
C08015=1096.997,119.920,437.540,176.580,16.613,152.226
C08016=1096.992,119.671,437.559,176.577,16.612,152.227
C08017=1096.986,119.422,437.578,176.574,16.611,152.227
C08018=1096.981,119.173,437.597,176.571,16.611,152.228
C08019=1096.975,118.924,437.617,176.568,16.611,152.228
C08020=1096.969,118.675,437.636,176.566,16.611,152.229
C08021=1096.964,118.425,437.656,176.563,16.610,152.229
C08022=1096.958,118.176,437.674,176.560,16.609,152.229
C08023=1096.953,117.927,437.694,176.558,16.609,152.230
C08024=1096.947,117.678,437.713,176.555,16.608,152.230
C08025=1096.942,117.429,437.732,176.552,16.608,152.231
C08026=1096.936,117.179,437.751,176.549,16.608,152.231
C08027=1096.931,116.930,437.770,176.546,16.607,152.232
C08028=1096.925,116.681,437.790,176.544,16.607,152.232
C08029=1096.920,116.432,437.808,176.541,16.606,152.233
C08030=1096.913,116.183,437.827,176.538,16.605,152.233
C08031=1096.908,115.933,437.846,176.536,16.605,152.234
C08032=1096.903,115.685,437.865,176.533,16.605,152.234
C08033=1096.897,115.435,437.884,176.530,16.604,152.234
C08034=1096.891,115.186,437.904,176.527,16.604,152.235
C08035=1096.886,114.937,437.923,176.525,16.603,152.235
C08036=1096.880,114.688,437.942,176.522,16.602,152.236
C08037=1096.875,114.438,437.961,176.519,16.602,152.236
C08038=1096.870,114.189,437.979,176.516,16.601,152.237
C08039=1096.864,113.940,437.998,176.514,16.601,152.237
C08040=1096.858,113.690,438.017,176.511,16.600,152.238
C08041=1096.852,113.441,438.036,176.509,16.600,152.238
C08042=1096.847,113.192,438.055,176.505,16.600,152.239
C08043=1096.841,112.943,438.074,176.503,16.599,152.239
C08044=1096.835,112.693,438.093,176.500,16.599,152.239
C08045=1096.830,112.445,438.112,176.497,16.598,152.240
C08046=1096.824,112.170,438.133,176.494,16.598,152.240
C08047=1096.818,111.895,438.153,176.492,16.597,152.241
C08048=1096.811,111.620,438.175,176.489,16.596,152.241
C08049=1096.805,111.345,438.195,176.486,16.596,152.242
C08050=1096.799,111.096,438.214,176.483,16.595,152.242
C08051=1096.793,110.847,438.232,176.481,16.595,152.243
C08052=1096.788,110.597,438.251,176.478,16.594,152.243
C08053=1096.782,110.348,438.270,176.475,16.593,152.243
C08054=1096.777,110.099,438.288,176.472,16.594,152.244
C08055=1096.771,109.850,438.308,176.469,16.593,152.244
C08056=1096.765,109.600,438.326,176.467,16.593,152.245
C08057=1096.760,109.351,438.344,176.464,16.592,152.245
C08058=1096.754,109.102,438.364,176.461,16.591,152.246
C08059=1096.748,108.853,438.382,176.459,16.591,152.246
C08060=1096.743,108.604,438.401,176.456,16.590,152.247
C08061=1096.737,108.354,438.420,176.454,16.590,152.247
C08062=1096.731,108.105,438.438,176.451,16.589,152.247
C08063=1096.726,107.856,438.457,176.448,16.588,152.248
C08064=1096.719,107.607,438.475,176.445,16.588,152.248
C08065=1096.714,107.358,438.494,176.442,16.588,152.249
C08066=1096.709,107.108,438.513,176.440,16.587,152.249
C08067=1096.703,106.859,438.531,176.437,16.587,152.250
C08068=1096.698,106.609,438.549,176.435,16.586,152.250
C08069=1096.691,106.360,438.568,176.432,16.586,152.250
C08070=1096.686,106.111,438.587,176.429,16.585,152.251
C08071=1096.680,105.862,438.605,176.427,16.584,152.251
C08072=1096.674,105.612,438.624,176.424,16.584,152.252
C08073=1096.670,105.363,438.642,176.422,16.583,152.252
C08074=1096.663,105.114,438.661,176.419,16.583,152.252
C08075=1096.658,104.865,438.680,176.416,16.582,152.253
C08076=1096.652,104.615,438.698,176.413,16.582,152.253
C08077=1096.647,104.367,438.717,176.410,16.581,152.254
C08078=1096.641,104.117,438.735,176.409,16.580,152.254
C08079=1096.636,103.868,438.753,176.406,16.579,152.254
C08080=1096.630,103.618,438.771,176.403,16.579,152.255
C08081=1096.624,103.370,438.790,176.400,16.578,152.255
C08082=1096.618,103.120,438.808,176.397,16.577,152.256
C08083=1096.613,102.871,438.827,176.395,16.577,152.256
C08084=1096.607,102.621,438.845,176.392,16.576,152.256
C08085=1096.602,102.373,438.864,176.390,16.576,152.257
C08086=1096.596,102.123,438.882,176.387,16.575,152.257
C08087=1096.591,101.874,438.901,176.385,16.575,152.258
C08088=1096.585,101.624,438.919,176.382,16.574,152.258
C08089=1096.580,101.375,438.937,176.379,16.573,152.258
C08090=1096.574,101.126,438.955,176.377,16.573,152.259
C08091=1096.569,100.877,438.974,176.374,16.572,152.259
C08092=1096.562,100.628,438.992,176.372,16.572,152.260
C08093=1096.556,100.378,439.010,176.369,16.571,152.260
C08094=1096.551,100.128,439.028,176.367,16.571,152.260
C08095=1096.545,99.879,439.047,176.364,16.570,152.261
C08096=1096.540,99.630,439.065,176.361,16.569,152.261
C08097=1096.534,99.381,439.084,176.359,16.569,152.262
C08098=1096.528,99.132,439.101,176.356,16.568,152.262
C08099=1096.522,98.882,439.119,176.354,16.567,152.262
C08100=1096.516,98.634,439.138,176.351,16.567,152.263
C08101=1096.511,98.384,439.156,176.349,16.566,152.263
C08102=1096.505,98.135,439.174,176.346,16.566,152.264
C08103=1096.500,97.885,439.191,176.343,16.565,152.264
C08104=1096.494,97.636,439.211,176.341,16.564,152.264
C08105=1096.489,97.387,439.228,176.338,16.563,152.265
C08106=1096.483,97.137,439.246,176.336,16.563,152.265
C08107=1096.478,96.889,439.265,176.333,16.562,152.266
C08108=1096.471,96.639,439.283,176.330,16.562,152.266
C08109=1096.466,96.390,439.300,176.328,16.561,152.266
C08110=1096.459,96.115,439.321,176.325,16.560,152.267
C08111=1096.453,95.841,439.340,176.323,16.560,152.267
C08112=1096.447,95.565,439.360,176.320,16.559,152.267
C08113=1096.441,95.291,439.380,176.317,16.558,152.268
C08114=1096.435,95.041,439.398,176.314,16.557,152.268
C08115=1096.430,94.792,439.416,176.311,16.557,152.269
C08116=1096.424,94.543,439.435,176.309,16.556,152.269
C08117=1096.418,94.294,439.452,176.307,16.556,152.269
C08118=1096.413,94.045,439.470,176.304,16.555,152.270
C08119=1096.407,93.795,439.488,176.302,16.554,152.270
C08120=1096.402,93.546,439.506,176.299,16.553,152.271
C08121=1096.396,93.296,439.524,176.297,16.553,152.271
C08122=1096.390,93.047,439.541,176.294,16.552,152.271
C08123=1096.384,92.798,439.560,176.292,16.552,152.272
C08124=1096.379,92.548,439.578,176.289,16.551,152.272
C08125=1096.374,92.299,439.596,176.286,16.550,152.272
C08126=1096.368,92.050,439.613,176.284,16.549,152.273
C08127=1096.362,91.801,439.631,176.281,16.549,152.273
C08128=1096.356,91.551,439.649,176.279,16.548,152.273
C08129=1096.352,91.302,439.667,176.276,16.547,152.274
C08130=1096.346,91.052,439.685,176.274,16.546,152.274
C08131=1096.340,90.803,439.702,176.271,16.546,152.274
C08132=1096.334,90.554,439.720,176.269,16.545,152.275
C08133=1096.328,90.305,439.738,176.266,16.544,152.275
C08134=1096.323,90.056,439.756,176.264,16.544,152.276
C08135=1096.317,89.806,439.773,176.261,16.543,152.276
C08136=1096.311,89.557,439.791,176.259,16.542,152.276
C08137=1096.306,89.308,439.809,176.256,16.542,152.277
C08138=1096.300,89.058,439.827,176.253,16.541,152.277
C08139=1096.294,88.809,439.844,176.251,16.540,152.277
C08140=1096.289,88.560,439.862,176.248,16.539,152.278
C08141=1096.282,88.310,439.880,176.246,16.539,152.278
C08142=1096.277,88.061,439.897,176.243,16.538,152.278
C08143=1096.271,87.812,439.915,176.241,16.538,152.279
C08144=1096.265,87.562,439.933,176.239,16.536,152.279
C08145=1096.260,87.313,439.950,176.236,16.536,152.280
C08146=1096.254,87.064,439.968,176.233,16.535,152.280
C08147=1096.248,86.814,439.985,176.232,16.535,152.280
C08148=1096.243,86.565,440.003,176.229,16.534,152.281
C08149=1096.237,86.316,440.020,176.227,16.533,152.281
C08150=1096.231,86.066,440.038,176.224,16.532,152.281
C08151=1096.226,85.817,440.056,176.222,16.532,152.282
C08152=1096.220,85.568,440.073,176.219,16.531,152.282
C08153=1096.215,85.319,440.091,176.217,16.530,152.282
C08154=1096.209,85.069,440.108,176.214,16.529,152.283
C08155=1096.203,84.820,440.126,176.212,16.529,152.283
C08156=1096.198,84.570,440.143,176.209,16.528,152.283
C08157=1096.192,84.321,440.161,176.207,16.527,152.284
C08158=1096.185,84.072,440.178,176.204,16.526,152.284
C08159=1096.180,83.822,440.195,176.202,16.525,152.284
C08160=1096.175,83.573,440.212,176.199,16.525,152.285
C08161=1096.169,83.324,440.230,176.197,16.524,152.285
C08162=1096.163,83.075,440.248,176.194,16.523,152.285
C08163=1096.158,82.825,440.266,176.192,16.522,152.286
C08164=1096.152,82.576,440.282,176.190,16.522,152.286
C08165=1096.147,82.327,440.300,176.187,16.521,152.286
C08166=1096.141,82.077,440.318,176.185,16.520,152.287
C08167=1096.136,81.827,440.335,176.182,16.519,152.287
C08168=1096.130,81.578,440.352,176.180,16.519,152.287
C08169=1096.124,81.329,440.370,176.177,16.518,152.288
C08170=1096.119,81.080,440.386,176.175,16.517,152.288
C08171=1096.112,80.830,440.404,176.173,16.516,152.288
C08172=1096.107,80.581,440.422,176.170,16.516,152.289
C08173=1096.102,80.332,440.438,176.168,16.514,152.289
C08174=1096.096,80.057,440.458,176.165,16.514,152.289
C08175=1096.089,79.783,440.477,176.163,16.513,152.290
C08176=1096.084,79.508,440.496,176.160,16.512,152.290
C08177=1096.077,79.233,440.515,176.157,16.511,152.290
C08178=1096.071,78.984,440.533,176.155,16.510,152.290
C08179=1096.066,78.734,440.549,176.152,16.509,152.291
C08180=1096.060,78.485,440.566,176.150,16.509,152.291
C08181=1096.055,78.236,440.583,176.147,16.508,152.292
C08182=1096.048,77.986,440.601,176.145,16.507,152.292
C08183=1096.043,77.737,440.619,176.143,16.506,152.292
C08184=1096.037,77.488,440.635,176.141,16.506,152.293
C08185=1096.031,77.239,440.653,176.138,16.504,152.293
C08186=1096.026,76.989,440.669,176.136,16.504,152.293
C08187=1096.020,76.740,440.686,176.133,16.503,152.293
C08188=1096.014,76.490,440.704,176.131,16.502,152.294
C08189=1096.009,76.241,440.721,176.128,16.501,152.294
C08190=1096.003,75.991,440.738,176.126,16.501,152.294
C08191=1095.997,75.742,440.755,176.124,16.499,152.295
C08192=1095.992,75.493,440.772,176.122,16.499,152.295
C08193=1095.986,75.244,440.789,176.119,16.498,152.295
C08194=1095.980,74.994,440.806,176.117,16.497,152.296
C08195=1095.974,74.745,440.824,176.114,16.496,152.296
C08196=1095.968,74.495,440.840,176.112,16.495,152.296
C08197=1095.963,74.246,440.857,176.109,16.495,152.297
C08198=1095.958,73.997,440.874,176.107,16.494,152.297
C08199=1095.952,73.747,440.891,176.105,16.493,152.297
C08200=1095.946,73.498,440.908,176.103,16.492,152.297
C08201=1095.941,73.248,440.925,176.100,16.491,152.298
C08202=1095.935,73.000,440.942,176.098,16.490,152.298
C08203=1095.930,72.750,440.959,176.095,16.489,152.298
C08204=1095.924,72.500,440.976,176.093,16.489,152.299
C08205=1095.918,72.252,440.993,176.091,16.488,152.299
C08206=1095.912,72.001,441.010,176.088,16.487,152.299
C08207=1095.906,71.752,441.026,176.087,16.486,152.299
C08208=1095.901,71.503,441.044,176.084,16.485,152.300
C08209=1095.896,71.253,441.060,176.082,16.484,152.300
C08210=1095.890,71.004,441.077,176.079,16.484,152.300
C08211=1095.884,70.755,441.094,176.077,16.483,152.301
C08212=1095.878,70.506,441.111,176.074,16.482,152.301
C08213=1095.873,70.256,441.127,176.072,16.481,152.301
C08214=1095.867,70.007,441.144,176.070,16.480,152.301
C08215=1095.861,69.758,441.161,176.068,16.479,152.302
C08216=1095.856,69.508,441.178,176.065,16.478,152.302
C08217=1095.850,69.259,441.194,176.063,16.478,152.302
C08218=1095.844,69.010,441.211,176.060,16.476,152.303
C08219=1095.839,68.760,441.228,176.058,16.476,152.303
C08220=1095.833,68.511,441.244,176.056,16.474,152.303
C08221=1095.828,68.261,441.261,176.054,16.474,152.303
C08222=1095.821,68.012,441.278,176.051,16.473,152.304
C08223=1095.816,67.763,441.295,176.049,16.472,152.304
C08224=1095.810,67.513,441.311,176.047,16.472,152.304
C08225=1095.805,67.264,441.328,176.044,16.470,152.305
C08226=1095.799,67.014,441.344,176.042,16.470,152.305
C08227=1095.794,66.765,441.362,176.040,16.468,152.305
C08228=1095.788,66.516,441.378,176.038,16.468,152.305
C08229=1095.782,66.267,441.395,176.035,16.467,152.306
C08230=1095.776,66.017,441.411,176.033,16.466,152.306
C08231=1095.770,65.768,441.428,176.030,16.465,152.306
C08232=1095.765,65.518,441.445,176.028,16.464,152.307
C08233=1095.759,65.269,441.461,176.026,16.463,152.307
C08234=1095.753,65.020,441.478,176.024,16.462,152.307
C08235=1095.748,64.770,441.495,176.021,16.461,152.307
C08236=1095.742,64.521,441.511,176.019,16.460,152.308
C08237=1095.737,64.271,441.528,176.017,16.460,152.308
C08238=1095.730,63.997,441.546,176.014,16.459,152.308
C08239=1095.724,63.722,441.564,176.012,16.458,152.309
C08240=1095.717,63.447,441.582,176.009,16.456,152.309
C08241=1095.710,63.172,441.600,176.007,16.456,152.309
C08242=1095.705,62.922,441.617,176.004,16.454,152.310
C08243=1095.699,62.673,441.633,176.003,16.454,152.310
C08244=1095.693,62.424,441.649,176.000,16.453,152.310
C08245=1095.687,62.174,441.666,175.998,16.452,152.310
C08246=1095.681,61.925,441.682,175.996,16.452,152.311
C08247=1095.676,61.675,441.698,175.993,16.450,152.311
C08248=1095.670,61.426,441.715,175.991,16.450,152.311
C08249=1095.664,61.176,441.732,175.988,16.448,152.311
C08250=1095.659,60.928,441.747,175.987,16.448,152.312
C08251=1095.653,60.678,441.764,175.984,16.446,152.312
C08252=1095.647,60.429,441.780,175.982,16.446,152.312
C08253=1095.641,60.179,441.796,175.979,16.444,152.313
C08254=1095.636,59.930,441.813,175.977,16.444,152.313
C08255=1095.630,59.680,441.829,175.976,16.443,152.313
C08256=1095.624,59.431,441.846,175.973,16.442,152.313
C08257=1095.618,59.182,441.862,175.971,16.441,152.314
C08258=1095.612,58.932,441.878,175.968,16.440,152.314
C08259=1095.606,58.683,441.894,175.966,16.439,152.314
C08260=1095.601,58.433,441.911,175.964,16.438,152.314
C08261=1095.595,58.184,441.927,175.962,16.437,152.315
C08262=1095.589,57.934,441.943,175.960,16.437,152.315
C08263=1095.583,57.685,441.959,175.957,16.435,152.315
C08264=1095.577,57.435,441.975,175.955,16.435,152.315
C08265=1095.572,57.187,441.991,175.953,16.433,152.316
C08266=1095.566,56.937,442.008,175.951,16.433,152.316
C08267=1095.561,56.688,442.024,175.948,16.431,152.316
C08268=1095.555,56.438,442.041,175.946,16.431,152.316
C08269=1095.549,56.188,442.056,175.944,16.430,152.317
C08270=1095.543,55.939,442.073,175.941,16.429,152.317
C08271=1095.537,55.690,442.089,175.940,16.428,152.317
C08272=1095.531,55.440,442.105,175.937,16.427,152.318
C08273=1095.526,55.192,442.121,175.935,16.426,152.318
C08274=1095.520,54.942,442.136,175.933,16.424,152.318
C08275=1095.515,54.692,442.153,175.931,16.424,152.318
C08276=1095.509,54.443,442.170,175.929,16.423,152.318
C08277=1095.503,54.193,442.186,175.926,16.422,152.319
C08278=1095.498,53.943,442.201,175.924,16.421,152.319
C08279=1095.492,53.695,442.217,175.922,16.420,152.319
C08280=1095.486,53.445,442.234,175.920,16.419,152.319
C08281=1095.481,53.195,442.249,175.917,16.418,152.320
C08282=1095.475,52.946,442.265,175.915,16.417,152.320
C08283=1095.469,52.697,442.282,175.913,16.416,152.320
C08284=1095.464,52.448,442.297,175.911,16.415,152.320
C08285=1095.458,52.198,442.313,175.909,16.414,152.321
C08286=1095.452,51.949,442.329,175.906,16.413,152.321
C08287=1095.446,51.699,442.346,175.904,16.412,152.321
C08288=1095.440,51.450,442.361,175.903,16.411,152.321
C08289=1095.436,51.201,442.378,175.900,16.410,152.322
C08290=1095.430,50.951,442.393,175.898,16.409,152.322
C08291=1095.424,50.701,442.409,175.895,16.408,152.322
C08292=1095.418,50.452,442.426,175.894,16.407,152.322
C08293=1095.413,50.203,442.441,175.891,16.405,152.322
C08294=1095.407,49.953,442.457,175.889,16.405,152.323
C08295=1095.402,49.703,442.473,175.887,16.404,152.323
C08296=1095.396,49.454,442.489,175.885,16.403,152.323
C08297=1095.390,49.205,442.505,175.883,16.402,152.323
C08298=1095.385,48.955,442.520,175.880,16.400,152.324
C08299=1095.379,48.706,442.537,175.878,16.400,152.324
C08300=1095.373,48.456,442.552,175.877,16.399,152.324
C08301=1095.368,48.207,442.568,175.874,16.397,152.324
C08302=1095.361,47.933,442.585,175.872,16.397,152.324
C08303=1095.355,47.657,442.602,175.870,16.395,152.325
C08304=1095.349,47.382,442.620,175.867,16.394,152.325
C08305=1095.342,47.107,442.637,175.865,16.393,152.325
C08306=1095.337,46.858,442.653,175.863,16.392,152.325
C08307=1095.331,46.608,442.669,175.861,16.391,152.326
C08308=1095.326,46.358,442.684,175.858,16.390,152.326
C08309=1095.320,46.110,442.700,175.856,16.389,152.326
C08310=1095.315,45.860,442.716,175.854,16.388,152.326
C08311=1095.309,45.610,442.732,175.852,16.387,152.327
C08312=1095.304,45.361,442.747,175.850,16.385,152.327
C08313=1095.298,45.112,442.764,175.847,16.384,152.327
C08314=1095.292,44.862,442.779,175.846,16.384,152.327
C08315=1095.287,44.613,442.795,175.844,16.382,152.327
C08316=1095.281,44.363,442.811,175.841,16.381,152.328
C08317=1095.275,44.113,442.826,175.839,16.380,152.328
C08318=1095.270,43.865,442.842,175.837,16.379,152.328
C08319=1095.264,43.615,442.857,175.835,16.378,152.328
C08320=1095.258,43.366,442.873,175.833,16.377,152.328
C08321=1095.253,43.116,442.888,175.831,16.376,152.329
C08322=1095.247,42.866,442.904,175.829,16.375,152.329
C08323=1095.241,42.617,442.920,175.826,16.374,152.329
C08324=1095.235,42.368,442.935,175.825,16.372,152.329
C08325=1095.230,42.118,442.950,175.823,16.372,152.329
C08326=1095.224,41.869,442.966,175.820,16.371,152.330
C08327=1095.219,41.619,442.982,175.818,16.369,152.330
C08328=1095.213,41.369,442.997,175.817,16.369,152.330
C08329=1095.206,41.120,443.013,175.814,16.367,152.330
C08330=1095.201,40.871,443.028,175.812,16.366,152.330
C08331=1095.196,40.621,443.044,175.810,16.365,152.331
C08332=1095.191,40.372,443.059,175.808,16.364,152.331
C08333=1095.184,40.123,443.074,175.806,16.363,152.331
C08334=1095.178,39.873,443.090,175.803,16.362,152.331
C08335=1095.173,39.624,443.105,175.801,16.361,152.332
C08336=1095.167,39.374,443.121,175.800,16.360,152.332
C08337=1095.161,39.125,443.136,175.797,16.359,152.332
C08338=1095.156,38.875,443.152,175.796,16.358,152.332
C08339=1095.150,38.625,443.167,175.793,16.356,152.332
C08340=1095.145,38.376,443.182,175.791,16.356,152.333
C08341=1095.138,38.127,443.198,175.789,16.355,152.333
C08342=1095.133,37.878,443.213,175.787,16.353,152.333
C08343=1095.128,37.628,443.229,175.785,16.352,152.333
C08344=1095.121,37.378,443.244,175.783,16.351,152.333
C08345=1095.116,37.129,443.259,175.780,16.350,152.334
C08346=1095.110,36.880,443.274,175.779,16.349,152.334
C08347=1095.104,36.630,443.290,175.776,16.348,152.334
C08348=1095.099,36.381,443.305,175.774,16.347,152.334
C08349=1095.093,36.131,443.320,175.773,16.346,152.334
C08350=1095.087,35.882,443.335,175.770,16.345,152.335
C08351=1095.081,35.632,443.350,175.768,16.344,152.335
C08352=1095.075,35.382,443.366,175.766,16.343,152.335
C08353=1095.069,35.134,443.381,175.764,16.342,152.335
C08354=1095.064,34.884,443.397,175.762,16.340,152.335
C08355=1095.058,34.635,443.411,175.760,16.340,152.336
C08356=1095.052,34.385,443.427,175.758,16.338,152.336
C08357=1095.047,34.136,443.442,175.756,16.337,152.336
C08358=1095.041,33.886,443.457,175.754,16.337,152.336
C08359=1095.035,33.636,443.472,175.752,16.335,152.336
C08360=1095.029,33.387,443.487,175.750,16.334,152.337
C08361=1095.024,33.137,443.502,175.748,16.333,152.337
C08362=1095.018,32.888,443.517,175.746,16.332,152.337
C08363=1095.012,32.638,443.533,175.744,16.331,152.337
C08364=1095.007,32.389,443.547,175.741,16.329,152.337
C08365=1095.001,32.139,443.563,175.740,16.328,152.338
C08366=1094.995,31.865,443.580,175.738,16.328,152.338
C08367=1094.988,31.590,443.596,175.735,16.326,152.338
C08368=1094.982,31.314,443.613,175.733,16.325,152.338
C08369=1094.976,31.040,443.629,175.731,16.324,152.338
C08370=1094.970,30.790,443.644,175.728,16.322,152.339
C08371=1094.964,30.541,443.659,175.726,16.322,152.339
C08372=1094.959,30.291,443.674,175.725,16.320,152.339
C08373=1094.953,30.042,443.689,175.722,16.319,152.339
C08374=1094.947,29.792,443.704,175.721,16.318,152.339
C08375=1094.942,29.543,443.719,175.719,16.317,152.340
C08376=1094.935,29.293,443.734,175.716,16.316,152.340
C08377=1094.930,29.044,443.749,175.714,16.315,152.340
C08378=1094.924,28.795,443.764,175.713,16.314,152.340
C08379=1094.919,28.545,443.779,175.710,16.312,152.340
C08380=1094.913,28.296,443.794,175.708,16.311,152.340
C08381=1094.907,28.046,443.810,175.707,16.311,152.341
C08382=1094.902,27.796,443.823,175.704,16.309,152.341
C08383=1094.895,27.547,443.838,175.702,16.308,152.341
C08384=1094.890,27.297,443.854,175.701,16.307,152.341
C08385=1094.884,27.048,443.868,175.698,16.306,152.341
C08386=1094.878,26.799,443.883,175.696,16.305,152.342
C08387=1094.873,26.549,443.899,175.695,16.303,152.342
C08388=1094.867,26.300,443.913,175.692,16.302,152.342
C08389=1094.861,26.050,443.927,175.690,16.301,152.342
C08390=1094.856,25.800,443.943,175.689,16.300,152.342
C08391=1094.849,25.551,443.958,175.686,16.299,152.342
C08392=1094.843,25.302,443.972,175.684,16.298,152.343
C08393=1094.838,25.052,443.988,175.683,16.297,152.343
C08394=1094.832,24.802,444.002,175.681,16.296,152.343
C08395=1094.826,24.553,444.016,175.678,16.294,152.343
C08396=1094.820,24.304,444.031,175.676,16.294,152.343
C08397=1094.815,24.054,444.046,175.675,16.293,152.343
C08398=1094.809,23.804,444.060,175.672,16.291,152.344
C08399=1094.803,23.555,444.075,175.671,16.290,152.344
C08400=1094.798,23.305,444.091,175.669,16.289,152.344
C08401=1094.792,23.056,444.105,175.666,16.288,152.344
C08402=1094.786,22.806,444.119,175.665,16.287,152.344
C08403=1094.780,22.557,444.134,175.663,16.286,152.345
C08404=1094.775,22.308,444.149,175.660,16.284,152.345
C08405=1094.769,22.057,444.163,175.658,16.283,152.345
C08406=1094.763,21.808,444.178,175.657,16.282,152.345
C08407=1094.757,21.560,444.193,175.654,16.281,152.345
C08408=1094.752,21.309,444.207,175.653,16.280,152.345
C08409=1094.746,21.060,444.222,175.651,16.279,152.346
C08410=1094.740,20.810,444.237,175.649,16.278,152.346
C08411=1094.734,20.561,444.251,175.647,16.276,152.346
C08412=1094.729,20.311,444.266,175.645,16.275,152.346
C08413=1094.723,20.062,444.281,175.643,16.274,152.346
C08414=1094.717,19.812,444.295,175.641,16.273,152.346
C08415=1094.711,19.563,444.310,175.639,16.272,152.346
C08416=1094.705,19.314,444.324,175.637,16.271,152.347
C08417=1094.701,19.064,444.339,175.635,16.269,152.347
C08418=1094.694,18.814,444.354,175.633,16.268,152.347
C08419=1094.689,18.565,444.368,175.631,16.267,152.347
C08420=1094.683,18.316,444.382,175.630,16.266,152.347
C08421=1094.677,18.065,444.396,175.627,16.265,152.348
C08422=1094.671,17.816,444.411,175.625,16.264,152.348
C08423=1094.665,17.567,444.425,175.624,16.263,152.348
C08424=1094.659,17.317,444.440,175.621,16.261,152.348
C08425=1094.654,17.068,444.455,175.620,16.260,152.348
C08426=1094.649,16.818,444.469,175.618,16.260,152.348
C08427=1094.642,16.569,444.484,175.616,16.258,152.349
C08428=1094.637,16.319,444.498,175.614,16.257,152.349
C08429=1094.631,16.070,444.512,175.612,16.256,152.349
C08430=1094.624,15.796,444.528,175.609,16.254,152.349
C08431=1094.618,15.523,444.544,175.608,16.253,152.349
C08432=1094.612,15.249,444.559,175.605,16.252,152.349
C08433=1094.606,14.976,444.575,175.603,16.251,152.350
C08434=1094.600,14.725,444.590,175.602,16.250,152.350
C08435=1094.595,14.476,444.604,175.599,16.248,152.350
C08436=1094.589,14.227,444.618,175.598,16.247,152.350
C08437=1094.583,13.977,444.633,175.596,16.246,152.350
C08438=1094.577,13.727,444.647,175.594,16.245,152.350
C08439=1094.571,13.479,444.661,175.592,16.243,152.351
C08440=1094.565,13.229,444.675,175.590,16.243,152.351
C08441=1094.559,12.980,444.690,175.588,16.242,152.351
C08442=1094.553,12.730,444.704,175.586,16.240,152.351
C08443=1094.547,12.480,444.718,175.584,16.239,152.351
C08444=1094.541,12.231,444.732,175.582,16.238,152.351
C08445=1094.536,11.981,444.746,175.580,16.237,152.352
C08446=1094.530,11.731,444.760,175.578,16.236,152.352
C08447=1094.524,11.482,444.775,175.576,16.235,152.352
C08448=1094.519,11.232,444.789,175.575,16.234,152.352
C08449=1094.512,10.983,444.804,175.573,16.233,152.352
C08450=1094.507,10.733,444.818,175.571,16.231,152.352
C08451=1094.501,10.484,444.831,175.569,16.230,152.353
C08452=1094.495,10.235,444.846,175.567,16.229,152.353
C08453=1094.489,9.985,444.860,175.565,16.228,152.353
C08454=1094.483,9.735,444.874,175.563,16.227,152.353
C08455=1094.477,9.486,444.888,175.561,16.226,152.353
C08456=1094.471,9.236,444.902,175.560,16.224,152.353
C08457=1094.466,8.986,444.916,175.558,16.224,152.354
C08458=1094.460,8.737,444.930,175.555,16.222,152.354
C08459=1094.454,8.488,444.944,175.554,16.221,152.354
C08460=1094.448,8.238,444.958,175.552,16.220,152.354
C08461=1094.442,7.988,444.972,175.549,16.218,152.354
C08462=1094.437,7.739,444.986,175.548,16.217,152.354
C08463=1094.431,7.490,445.001,175.546,16.217,152.354
C08464=1094.425,7.239,445.015,175.544,16.215,152.355
C08465=1094.420,6.990,445.029,175.542,16.214,152.355
C08466=1094.413,6.741,445.042,175.540,16.213,152.355
C08467=1094.408,6.492,445.057,175.538,16.212,152.355
C08468=1094.402,6.242,445.070,175.537,16.211,152.355
C08469=1094.396,5.992,445.085,175.534,16.209,152.355
C08470=1094.391,5.742,445.099,175.532,16.208,152.356
C08471=1094.385,5.493,445.112,175.531,16.207,152.356
C08472=1094.379,5.244,445.126,175.529,16.206,152.356
C08473=1094.373,4.994,445.140,175.527,16.204,152.356
C08474=1094.367,4.744,445.155,175.525,16.204,152.356
C08475=1094.362,4.495,445.168,175.523,16.202,152.356
C08476=1094.356,4.245,445.182,175.522,16.201,152.356
C08477=1094.350,3.996,445.196,175.520,16.200,152.356
C08478=1094.344,3.746,445.209,175.517,16.199,152.357
C08479=1094.339,3.497,445.223,175.516,16.198,152.357
C08480=1094.332,3.247,445.238,175.514,16.197,152.357
C08481=1094.327,2.997,445.252,175.513,16.195,152.357
C08482=1094.321,2.748,445.265,175.510,16.194,152.357
C08483=1094.315,2.498,445.279,175.508,16.193,152.357
C08484=1094.310,2.249,445.293,175.507,16.192,152.357
C08485=1094.304,1.999,445.307,175.505,16.191,152.358
C08486=1094.299,1.750,445.321,175.503,16.189,152.358
C08487=1094.292,1.500,445.334,175.501,16.188,152.358
C08488=1094.287,1.250,445.348,175.499,16.187,152.358
C08489=1094.281,1.001,445.362,175.498,16.186,152.358
C08490=1094.276,0.751,445.376,175.495,16.184,152.358
C08491=1094.269,0.502,445.389,175.494,16.183,152.358
C08492=1094.264,0.252,445.403,175.492,16.182,152.359
C08493=1094.258,0.003,445.417,175.490,16.181,152.359
C08494=1094.252,-0.269,445.432,175.488,16.179,152.359
C08495=1094.246,-0.540,445.447,175.486,16.178,152.359
C08496=1094.239,-0.812,445.462,175.483,16.177,152.359
C08497=1094.233,-1.083,445.477,175.482,16.176,152.359
C08498=1094.228,-1.333,445.491,175.480,16.175,152.360
C08499=1094.222,-1.582,445.504,175.479,16.174,152.360
C08500=1094.216,-1.832,445.518,175.476,16.172,152.360
C08501=1094.211,-2.081,445.532,175.475,16.171,152.360
C08502=1094.205,-2.331,445.546,175.473,16.170,152.360
C08503=1094.198,-2.581,445.559,175.471,16.169,152.360
C08504=1094.193,-2.831,445.573,175.469,16.167,152.360
C08505=1094.188,-3.080,445.587,175.467,16.166,152.360
C08506=1094.182,-3.330,445.600,175.466,16.165,152.361
C08507=1094.176,-3.580,445.613,175.464,16.164,152.361
C08508=1094.170,-3.829,445.627,175.462,16.163,152.361
C08509=1094.164,-4.078,445.641,175.460,16.161,152.361
C08510=1094.159,-4.328,445.654,175.458,16.160,152.361
C08511=1094.153,-4.577,445.668,175.456,16.159,152.361
C08512=1094.147,-4.827,445.682,175.455,16.158,152.361
C08513=1094.141,-5.076,445.695,175.453,16.157,152.362
C08514=1094.135,-5.326,445.709,175.451,16.155,152.362
C08515=1094.129,-5.576,445.722,175.449,16.154,152.362
C08516=1094.124,-5.826,445.735,175.447,16.153,152.362
C08517=1094.117,-6.075,445.749,175.445,16.152,152.362
C08518=1094.112,-6.325,445.763,175.444,16.151,152.362
C08519=1094.106,-6.574,445.776,175.441,16.149,152.362
C08520=1094.100,-6.823,445.789,175.440,16.149,152.363
C08521=1094.094,-7.073,445.802,175.438,16.148,152.363
C08522=1094.088,-7.323,445.816,175.436,16.146,152.363
C08523=1094.083,-7.572,445.829,175.435,16.145,152.363
C08524=1094.076,-7.822,445.843,175.432,16.144,152.363
C08525=1094.071,-8.072,445.856,175.430,16.143,152.363
C08526=1094.065,-8.321,445.869,175.429,16.142,152.363
C08527=1094.060,-8.571,445.883,175.427,16.141,152.364
C08528=1094.053,-8.820,445.896,175.426,16.139,152.364
C08529=1094.048,-9.069,445.910,175.423,16.138,152.364
C08530=1094.042,-9.319,445.923,175.421,16.137,152.364
C08531=1094.037,-9.569,445.936,175.420,16.136,152.364
C08532=1094.030,-9.818,445.950,175.418,16.135,152.364
C08533=1094.024,-10.068,445.962,175.417,16.133,152.364
C08534=1094.019,-10.318,445.976,175.414,16.132,152.364
C08535=1094.013,-10.567,445.989,175.412,16.131,152.365
C08536=1094.007,-10.816,446.003,175.411,16.130,152.365
C08537=1094.001,-11.066,446.016,175.409,16.129,152.365
C08538=1093.996,-11.316,446.030,175.407,16.128,152.365
C08539=1093.990,-11.565,446.043,175.406,16.126,152.365
C08540=1093.984,-11.815,446.056,175.403,16.125,152.365
C08541=1093.978,-12.065,446.069,175.402,16.124,152.366
C08542=1093.972,-12.314,446.082,175.400,16.123,152.366
C08543=1093.967,-12.564,446.096,175.398,16.122,152.366
C08544=1093.961,-12.813,446.109,175.397,16.121,152.366
C08545=1093.955,-13.063,446.122,175.394,16.119,152.366
C08546=1093.949,-13.313,446.136,175.393,16.118,152.366
C08547=1093.943,-13.562,446.149,175.391,16.117,152.366
C08548=1093.938,-13.812,446.162,175.389,16.116,152.366
C08549=1093.932,-14.061,446.175,175.388,16.115,152.366
C08550=1093.926,-14.311,446.188,175.386,16.114,152.367
C08551=1093.920,-14.561,446.202,175.384,16.112,152.367
C08552=1093.914,-14.810,446.215,175.382,16.111,152.367
C08553=1093.908,-15.060,446.227,175.380,16.109,152.367
C08554=1093.903,-15.309,446.241,175.379,16.109,152.367
C08555=1093.897,-15.559,446.253,175.377,16.108,152.367
C08556=1093.891,-15.808,446.267,175.375,16.106,152.367
C08557=1093.885,-16.058,446.279,175.373,16.105,152.368
C08558=1093.878,-16.328,446.294,175.371,16.104,152.368
C08559=1093.872,-16.598,446.308,175.369,16.103,152.368
C08560=1093.866,-16.868,446.322,175.367,16.101,152.368
C08561=1093.860,-17.138,446.336,175.365,16.100,152.368
C08562=1093.854,-17.388,446.349,175.364,16.099,152.368
C08563=1093.847,-17.637,446.362,175.362,16.098,152.368
C08564=1093.842,-17.887,446.375,175.360,16.097,152.369
C08565=1093.836,-18.137,446.389,175.359,16.096,152.369
C08566=1093.830,-18.387,446.401,175.356,16.094,152.369
C08567=1093.825,-18.635,446.414,175.355,16.093,152.369
C08568=1093.819,-18.885,446.427,175.353,16.092,152.369
C08569=1093.813,-19.135,446.440,175.351,16.091,152.369
C08570=1093.807,-19.384,446.453,175.350,16.090,152.369
C08571=1093.801,-19.634,446.466,175.348,16.089,152.369
C08572=1093.795,-19.884,446.479,175.346,16.087,152.370
C08573=1093.789,-20.133,446.492,175.344,16.086,152.370
C08574=1093.784,-20.383,446.505,175.342,16.085,152.370
C08575=1093.778,-20.633,446.518,175.341,16.084,152.370
C08576=1093.772,-20.882,446.531,175.339,16.083,152.370
C08577=1093.766,-21.131,446.543,175.337,16.082,152.370
C08578=1093.760,-21.381,446.557,175.336,16.081,152.370
C08579=1093.754,-21.630,446.569,175.333,16.079,152.371
C08580=1093.748,-21.880,446.582,175.331,16.078,152.371
C08581=1093.743,-22.130,446.596,175.330,16.077,152.371
C08582=1093.737,-22.380,446.608,175.328,16.076,152.371
C08583=1093.731,-22.630,446.621,175.327,16.075,152.371
C08584=1093.725,-22.878,446.634,175.325,16.074,152.371
C08585=1093.719,-23.128,446.646,175.323,16.072,152.371
C08586=1093.714,-23.378,446.659,175.322,16.072,152.372
C08587=1093.707,-23.627,446.672,175.319,16.070,152.372
C08588=1093.702,-23.878,446.685,175.318,16.069,152.372
C08589=1093.696,-24.127,446.698,175.316,16.068,152.372
C08590=1093.691,-24.376,446.711,175.314,16.067,152.372
C08591=1093.685,-24.626,446.723,175.313,16.065,152.372
C08592=1093.679,-24.876,446.736,175.311,16.064,152.372
C08593=1093.673,-25.126,446.748,175.309,16.064,152.372
C08594=1093.667,-25.375,446.761,175.308,16.062,152.373
C08595=1093.661,-25.624,446.774,175.305,16.061,152.373
C08596=1093.656,-25.874,446.786,175.304,16.060,152.373
C08597=1093.650,-26.124,446.799,175.302,16.058,152.373
C08598=1093.644,-26.373,446.813,175.300,16.057,152.373
C08599=1093.638,-26.623,446.825,175.299,16.056,152.373
C08600=1093.633,-26.872,446.837,175.297,16.055,152.373
C08601=1093.627,-27.122,446.850,175.295,16.054,152.373
C08602=1093.621,-27.372,446.863,175.294,16.053,152.374
C08603=1093.615,-27.621,446.876,175.291,16.051,152.374
C08604=1093.608,-27.871,446.888,175.290,16.050,152.374
C08605=1093.603,-28.120,446.900,175.288,16.050,152.374
C08606=1093.597,-28.370,446.912,175.286,16.048,152.374
C08607=1093.591,-28.619,446.926,175.285,16.047,152.374
C08608=1093.585,-28.869,446.938,175.283,16.046,152.374
C08609=1093.579,-29.119,446.951,175.281,16.045,152.374
C08610=1093.573,-29.369,446.963,175.280,16.044,152.375
C08611=1093.568,-29.618,446.976,175.278,16.043,152.375
C08612=1093.562,-29.868,446.988,175.276,16.042,152.375
C08613=1093.556,-30.117,447.001,175.274,16.040,152.375
C08614=1093.550,-30.367,447.014,175.272,16.039,152.375
C08615=1093.544,-30.616,447.026,175.271,16.038,152.375
C08616=1093.538,-30.866,447.038,175.269,16.037,152.376
C08617=1093.532,-31.116,447.051,175.267,16.036,152.376
C08618=1093.526,-31.366,447.063,175.266,16.035,152.376
C08619=1093.520,-31.616,447.076,175.264,16.034,152.376
C08620=1093.515,-31.865,447.088,175.262,16.033,152.376
C08621=1093.509,-32.115,447.100,175.261,16.032,152.376
C08622=1093.502,-32.383,447.114,175.258,16.030,152.376
C08623=1093.495,-32.653,447.128,175.257,16.029,152.376
C08624=1093.490,-32.922,447.141,175.255,16.028,152.377
C08625=1093.483,-33.191,447.154,175.253,16.027,152.377
C08626=1093.478,-33.441,447.167,175.251,16.026,152.377
C08627=1093.472,-33.691,447.179,175.249,16.024,152.377
C08628=1093.466,-33.940,447.191,175.247,16.023,152.377
C08629=1093.460,-34.189,447.204,175.246,16.022,152.377
C08630=1093.454,-34.439,447.216,175.244,16.021,152.377
C08631=1093.448,-34.689,447.228,175.243,16.020,152.377
C08632=1093.443,-34.938,447.241,175.241,16.019,152.378
C08633=1093.437,-35.188,447.253,175.239,16.018,152.378
C08634=1093.431,-35.438,447.266,175.238,16.017,152.378
C08635=1093.425,-35.687,447.278,175.236,16.015,152.378
C08636=1093.419,-35.937,447.290,175.234,16.014,152.378
C08637=1093.413,-36.187,447.303,175.233,16.013,152.378
C08638=1093.408,-36.436,447.315,175.231,16.013,152.378
C08639=1093.402,-36.686,447.327,175.229,16.011,152.379
C08640=1093.395,-36.935,447.339,175.227,16.010,152.379
C08641=1093.390,-37.185,447.352,175.225,16.008,152.379
C08642=1093.384,-37.435,447.364,175.224,16.007,152.379
C08643=1093.378,-37.684,447.377,175.222,16.006,152.379
C08644=1093.373,-37.934,447.389,175.220,16.005,152.379
C08645=1093.367,-38.183,447.401,175.219,16.004,152.379
C08646=1093.360,-38.433,447.413,175.217,16.003,152.379
C08647=1093.355,-38.683,447.425,175.215,16.002,152.380
C08648=1093.349,-38.933,447.437,175.214,16.001,152.380
C08649=1093.342,-39.182,447.449,175.212,16.000,152.380
C08650=1093.337,-39.432,447.462,175.210,15.999,152.380
C08651=1093.331,-39.681,447.474,175.209,15.998,152.380
C08652=1093.325,-39.931,447.486,175.207,15.997,152.380
C08653=1093.319,-40.180,447.498,175.205,15.996,152.380
C08654=1093.313,-40.430,447.511,175.204,15.995,152.381
C08655=1093.307,-40.680,447.522,175.202,15.994,152.381
C08656=1093.302,-40.929,447.534,175.200,15.992,152.381
C08657=1093.296,-41.179,447.547,175.198,15.991,152.381
C08658=1093.289,-41.429,447.559,175.196,15.990,152.381
C08659=1093.284,-41.678,447.571,175.194,15.989,152.381
C08660=1093.277,-41.928,447.583,175.193,15.988,152.381
C08661=1093.272,-42.178,447.595,175.191,15.987,152.382
C08662=1093.266,-42.427,447.607,175.190,15.986,152.382
C08663=1093.260,-42.677,447.619,175.188,15.985,152.382
C08664=1093.254,-42.927,447.631,175.186,15.984,152.382
C08665=1093.248,-43.176,447.644,175.185,15.983,152.382
C08666=1093.242,-43.426,447.655,175.183,15.981,152.382
C08667=1093.236,-43.676,447.667,175.181,15.980,152.382
C08668=1093.230,-43.925,447.679,175.179,15.980,152.383
C08669=1093.224,-44.175,447.692,175.178,15.978,152.383
C08670=1093.218,-44.424,447.702,175.176,15.977,152.383
C08671=1093.213,-44.674,447.715,175.175,15.976,152.383
C08672=1093.207,-44.924,447.728,175.173,15.975,152.383
C08673=1093.201,-45.174,447.738,175.171,15.974,152.383
C08674=1093.195,-45.423,447.751,175.170,15.973,152.383
C08675=1093.189,-45.672,447.763,175.168,15.972,152.383
C08676=1093.183,-45.922,447.775,175.166,15.971,152.384
C08677=1093.177,-46.173,447.787,175.164,15.970,152.384
C08678=1093.171,-46.422,447.799,175.163,15.969,152.384
C08679=1093.166,-46.671,447.811,175.161,15.968,152.384
C08680=1093.160,-46.921,447.822,175.160,15.967,152.384
C08681=1093.154,-47.171,447.835,175.158,15.966,152.384
C08682=1093.148,-47.420,447.846,175.156,15.965,152.384
C08683=1093.142,-47.670,447.858,175.155,15.964,152.385
C08684=1093.136,-47.920,447.870,175.153,15.963,152.385
C08685=1093.130,-48.169,447.882,175.151,15.961,152.385
C08686=1093.124,-48.438,447.895,175.149,15.960,152.385
C08687=1093.117,-48.708,447.908,175.147,15.959,152.385
C08688=1093.111,-48.977,447.920,175.145,15.958,152.385
C08689=1093.105,-49.247,447.933,175.144,15.957,152.385
C08690=1093.099,-49.497,447.944,175.142,15.956,152.385
C08691=1093.093,-49.746,447.957,175.140,15.955,152.386
C08692=1093.088,-49.997,447.968,175.139,15.954,152.386
C08693=1093.082,-50.245,447.980,175.137,15.953,152.386
C08694=1093.076,-50.495,447.993,175.136,15.951,152.386
C08695=1093.070,-50.745,448.003,175.134,15.951,152.386
C08696=1093.063,-50.994,448.015,175.132,15.950,152.386
C08697=1093.057,-51.245,448.027,175.130,15.948,152.387
C08698=1093.052,-51.494,448.039,175.129,15.947,152.387
C08699=1093.045,-51.744,448.050,175.127,15.947,152.387
C08700=1093.039,-51.993,448.062,175.125,15.945,152.387
C08701=1093.033,-52.243,448.074,175.124,15.944,152.387
C08702=1093.028,-52.492,448.085,175.122,15.944,152.387
C08703=1093.021,-52.742,448.097,175.120,15.942,152.387
C08704=1093.015,-52.992,448.109,175.119,15.941,152.388
C08705=1093.009,-53.241,448.121,175.117,15.941,152.388
C08706=1093.003,-53.491,448.132,175.115,15.939,152.388
C08707=1092.997,-53.740,448.143,175.114,15.938,152.388
C08708=1092.991,-53.991,448.155,175.112,15.938,152.388
C08709=1092.985,-54.240,448.167,175.110,15.937,152.388
C08710=1092.979,-54.490,448.178,175.108,15.935,152.388
C08711=1092.972,-54.739,448.190,175.107,15.935,152.389
C08712=1092.967,-54.989,448.201,175.105,15.934,152.389
C08713=1092.961,-55.239,448.213,175.103,15.932,152.389
C08714=1092.955,-55.488,448.224,175.101,15.932,152.389
C08715=1092.949,-55.738,448.236,175.100,15.931,152.389
C08716=1092.943,-55.988,448.248,175.098,15.929,152.389
C08717=1092.937,-56.238,448.259,175.096,15.929,152.390
C08718=1092.931,-56.487,448.271,175.095,15.928,152.390
C08719=1092.925,-56.737,448.282,175.093,15.926,152.390
C08720=1092.919,-56.986,448.294,175.091,15.926,152.390
C08721=1092.913,-57.236,448.305,175.090,15.925,152.390
C08722=1092.907,-57.486,448.316,175.088,15.923,152.390
C08723=1092.901,-57.735,448.328,175.086,15.922,152.390
C08724=1092.896,-57.985,448.340,175.085,15.922,152.391
C08725=1092.889,-58.235,448.351,175.084,15.921,152.391
C08726=1092.883,-58.484,448.362,175.082,15.920,152.391
C08727=1092.877,-58.734,448.374,175.080,15.919,152.391
C08728=1092.871,-58.983,448.385,175.079,15.918,152.391
C08729=1092.865,-59.234,448.397,175.077,15.917,152.391
C08730=1092.860,-59.483,448.408,175.075,15.916,152.392
C08731=1092.853,-59.733,448.420,175.074,15.915,152.392
C08732=1092.847,-59.982,448.431,175.072,15.914,152.392
C08733=1092.841,-60.232,448.442,175.070,15.913,152.392
C08734=1092.835,-60.482,448.454,175.068,15.912,152.392
C08735=1092.830,-60.731,448.465,175.067,15.911,152.392
C08736=1092.823,-60.981,448.476,175.065,15.910,152.393
C08737=1092.817,-61.230,448.488,175.063,15.909,152.393
C08738=1092.811,-61.480,448.499,175.062,15.908,152.393
C08739=1092.805,-61.730,448.510,175.060,15.907,152.393
C08740=1092.800,-61.980,448.522,175.058,15.906,152.393
C08741=1092.794,-62.229,448.533,175.057,15.905,152.393
C08742=1092.788,-62.479,448.544,175.055,15.904,152.394
C08743=1092.782,-62.729,448.556,175.053,15.903,152.394
C08744=1092.776,-62.978,448.566,175.052,15.903,152.394
C08745=1092.769,-63.228,448.578,175.050,15.902,152.394
C08746=1092.764,-63.478,448.590,175.049,15.901,152.394
C08747=1092.758,-63.727,448.601,175.047,15.900,152.394
C08748=1092.752,-63.977,448.612,175.045,15.899,152.394
C08749=1092.746,-64.226,448.624,175.044,15.898,152.395
C08750=1092.740,-64.498,448.635,175.042,15.897,152.395
C08751=1092.733,-64.768,448.648,175.040,15.896,152.395
C08752=1092.727,-65.039,448.660,175.039,15.895,152.395
C08753=1092.720,-65.309,448.672,175.036,15.893,152.395
C08754=1092.714,-65.560,448.683,175.035,15.893,152.395
C08755=1092.708,-65.809,448.694,175.034,15.892,152.395
C08756=1092.703,-66.059,448.705,175.032,15.891,152.396
C08757=1092.696,-66.309,448.716,175.030,15.890,152.396
C08758=1092.691,-66.558,448.729,175.028,15.889,152.396
C08759=1092.685,-66.808,448.740,175.027,15.888,152.396
C08760=1092.679,-67.058,448.751,175.025,15.887,152.396
C08761=1092.673,-67.307,448.762,175.023,15.886,152.396
C08762=1092.667,-67.557,448.773,175.022,15.885,152.397
C08763=1092.661,-67.807,448.784,175.020,15.884,152.397
C08764=1092.655,-68.056,448.795,175.018,15.883,152.397
C08765=1092.649,-68.306,448.807,175.017,15.882,152.397
C08766=1092.643,-68.555,448.817,175.016,15.882,152.397
C08767=1092.637,-68.805,448.828,175.014,15.881,152.397
C08768=1092.632,-69.055,448.840,175.012,15.880,152.398
C08769=1092.626,-69.305,448.851,175.010,15.879,152.398
C08770=1092.620,-69.554,448.862,175.009,15.878,152.398
C08771=1092.614,-69.804,448.873,175.007,15.877,152.398
C08772=1092.608,-70.054,448.884,175.005,15.876,152.398
C08773=1092.602,-70.304,448.895,175.004,15.875,152.398
C08774=1092.597,-70.553,448.906,175.002,15.874,152.399
C08775=1092.590,-70.803,448.917,175.000,15.873,152.399
C08776=1092.585,-71.053,448.928,174.999,15.872,152.399
C08777=1092.579,-71.302,448.939,174.998,15.872,152.399
C08778=1092.573,-71.552,448.950,174.996,15.870,152.399
C08779=1092.567,-71.802,448.961,174.994,15.869,152.399
C08780=1092.561,-72.051,448.972,174.992,15.869,152.399
C08781=1092.555,-72.301,448.983,174.991,15.867,152.400
C08782=1092.550,-72.550,448.994,174.989,15.866,152.400
C08783=1092.543,-72.801,449.005,174.987,15.866,152.400
C08784=1092.537,-73.050,449.016,174.986,15.865,152.400
C08785=1092.532,-73.299,449.027,174.985,15.864,152.400
C08786=1092.526,-73.549,449.037,174.983,15.863,152.400
C08787=1092.520,-73.799,449.049,174.981,15.862,152.400
C08788=1092.515,-74.049,449.060,174.980,15.861,152.401
C08789=1092.508,-74.298,449.070,174.978,15.860,152.401
C08790=1092.502,-74.548,449.081,174.976,15.859,152.401
C08791=1092.496,-74.798,449.093,174.974,15.858,152.401
C08792=1092.490,-75.047,449.103,174.973,15.857,152.401
C08793=1092.485,-75.297,449.114,174.972,15.857,152.401
C08794=1092.478,-75.547,449.126,174.970,15.856,152.402
C08795=1092.472,-75.796,449.136,174.968,15.855,152.402
C08796=1092.466,-76.046,449.147,174.967,15.854,152.402
C08797=1092.460,-76.296,449.158,174.965,15.854,152.402
C08798=1092.454,-76.546,449.168,174.963,15.852,152.402
C08799=1092.448,-76.795,449.179,174.961,15.852,152.403
C08800=1092.443,-77.045,449.190,174.960,15.851,152.403
C08801=1092.436,-77.295,449.201,174.959,15.851,152.403
C08802=1092.431,-77.545,449.212,174.957,15.849,152.403
C08803=1092.424,-77.794,449.222,174.955,15.848,152.403
C08804=1092.418,-78.043,449.233,174.953,15.848,152.403
C08805=1092.412,-78.293,449.244,174.952,15.846,152.404
C08806=1092.407,-78.544,449.255,174.950,15.846,152.404
C08807=1092.401,-78.793,449.265,174.949,15.845,152.404
C08808=1092.394,-79.042,449.276,174.947,15.845,152.404
C08809=1092.388,-79.292,449.287,174.946,15.843,152.404
C08810=1092.382,-79.542,449.298,174.944,15.843,152.404
C08811=1092.377,-79.791,449.309,174.942,15.842,152.405
C08812=1092.371,-80.042,449.319,174.940,15.841,152.405
C08813=1092.365,-80.291,449.329,174.939,15.840,152.405
C08814=1092.358,-80.564,449.341,174.937,15.839,152.405
C08815=1092.351,-80.838,449.353,174.935,15.838,152.405
C08816=1092.345,-81.110,449.365,174.933,15.837,152.406
C08817=1092.338,-81.383,449.377,174.931,15.837,152.406
C08818=1092.332,-81.633,449.387,174.931,15.836,152.406
C08819=1092.326,-81.882,449.397,174.929,15.835,152.406
C08820=1092.320,-82.132,449.408,174.927,15.834,152.406
C08821=1092.314,-82.382,449.419,174.925,15.834,152.407
C08822=1092.307,-82.631,449.429,174.924,15.832,152.407
C08823=1092.302,-82.881,449.440,174.922,15.832,152.407
C08824=1092.295,-83.130,449.450,174.921,15.832,152.407
C08825=1092.289,-83.381,449.461,174.919,15.831,152.407
C08826=1092.283,-83.630,449.472,174.917,15.830,152.408
C08827=1092.277,-83.880,449.482,174.915,15.829,152.408
C08828=1092.271,-84.129,449.492,174.914,15.828,152.408
C08829=1092.265,-84.379,449.504,174.913,15.828,152.408
C08830=1092.259,-84.629,449.513,174.911,15.827,152.408
C08831=1092.253,-84.879,449.524,174.909,15.826,152.408
C08832=1092.246,-85.128,449.534,174.907,15.825,152.409
C08833=1092.241,-85.378,449.545,174.905,15.824,152.409
C08834=1092.235,-85.628,449.556,174.905,15.824,152.409
C08835=1092.228,-85.877,449.566,174.903,15.823,152.409
C08836=1092.223,-86.127,449.577,174.901,15.822,152.409
C08837=1092.216,-86.377,449.587,174.899,15.821,152.410
C08838=1092.211,-86.626,449.597,174.897,15.821,152.410
C08839=1092.205,-86.877,449.608,174.897,15.820,152.410
C08840=1092.198,-87.126,449.618,174.895,15.820,152.410
C08841=1092.192,-87.376,449.629,174.893,15.818,152.410
C08842=1092.186,-87.625,449.639,174.891,15.818,152.411
C08843=1092.180,-87.875,449.650,174.889,15.817,152.411
C08844=1092.174,-88.124,449.660,174.888,15.816,152.411
C08845=1092.168,-88.375,449.670,174.887,15.816,152.411
C08846=1092.162,-88.624,449.681,174.885,15.815,152.411
C08847=1092.156,-88.874,449.691,174.883,15.814,152.411
C08848=1092.150,-89.124,449.702,174.881,15.813,152.412
C08849=1092.144,-89.373,449.712,174.880,15.813,152.412
C08850=1092.138,-89.623,449.722,174.878,15.812,152.412
C08851=1092.132,-89.872,449.732,174.877,15.811,152.412
C08852=1092.126,-90.123,449.743,174.875,15.810,152.412
C08853=1092.119,-90.372,449.753,174.874,15.810,152.413
C08854=1092.114,-90.622,449.764,174.872,15.809,152.413
C08855=1092.108,-90.872,449.774,174.870,15.808,152.413
C08856=1092.102,-91.121,449.785,174.869,15.807,152.413
C08857=1092.096,-91.371,449.795,174.867,15.807,152.413
C08858=1092.090,-91.620,449.805,174.866,15.807,152.414
C08859=1092.084,-91.870,449.815,174.864,15.805,152.414
C08860=1092.078,-92.120,449.825,174.862,15.805,152.414
C08861=1092.072,-92.370,449.836,174.860,15.804,152.414
C08862=1092.065,-92.620,449.846,174.859,15.804,152.414
C08863=1092.060,-92.870,449.856,174.858,15.803,152.415
C08864=1092.053,-93.119,449.867,174.856,15.802,152.415
C08865=1092.048,-93.369,449.877,174.854,15.801,152.415
C08866=1092.042,-93.618,449.887,174.852,15.800,152.415
C08867=1092.036,-93.868,449.897,174.851,15.800,152.415
C08868=1092.030,-94.117,449.908,174.849,15.799,152.416
C08869=1092.024,-94.367,449.918,174.848,15.799,152.416
C08870=1092.018,-94.617,449.928,174.846,15.797,152.416
C08871=1092.012,-94.867,449.938,174.845,15.797,152.416
C08872=1092.006,-95.117,449.948,174.843,15.797,152.416
C08873=1092.000,-95.366,449.959,174.841,15.795,152.417
C08874=1091.994,-95.617,449.969,174.839,15.795,152.417
C08875=1091.988,-95.866,449.979,174.839,15.794,152.417
C08876=1091.982,-96.116,449.989,174.837,15.794,152.417
C08877=1091.976,-96.365,450.000,174.835,15.793,152.417
C08878=1091.969,-96.641,450.010,174.833,15.792,152.418
C08879=1091.963,-96.915,450.021,174.831,15.791,152.418
C08880=1091.957,-97.190,450.033,174.829,15.790,152.418
C08881=1091.950,-97.466,450.044,174.828,15.790,152.418
C08882=1091.944,-97.716,450.054,174.827,15.789,152.418
C08883=1091.938,-97.965,450.064,174.825,15.789,152.419
C08884=1091.932,-98.216,450.075,174.823,15.788,152.419
C08885=1091.926,-98.466,450.084,174.822,15.788,152.419
C08886=1091.919,-98.715,450.095,174.820,15.787,152.419
C08887=1091.913,-98.965,450.104,174.818,15.786,152.419
C08888=1091.907,-99.214,450.115,174.816,15.785,152.420
C08889=1091.901,-99.464,450.125,174.815,15.785,152.420
C08890=1091.895,-99.714,450.134,174.814,15.784,152.420
C08891=1091.889,-99.963,450.145,174.812,15.784,152.420
C08892=1091.883,-100.213,450.155,174.810,15.783,152.421
C08893=1091.877,-100.463,450.164,174.809,15.783,152.421
C08894=1091.870,-100.712,450.174,174.807,15.782,152.421
C08895=1091.865,-100.962,450.185,174.805,15.781,152.421
C08896=1091.859,-101.212,450.194,174.804,15.781,152.421
C08897=1091.852,-101.462,450.204,174.802,15.780,152.422
C08898=1091.847,-101.711,450.215,174.801,15.779,152.422
C08899=1091.841,-101.961,450.224,174.799,15.778,152.422
C08900=1091.834,-102.211,450.234,174.798,15.778,152.422
C08901=1091.828,-102.460,450.244,174.796,15.778,152.423
C08902=1091.822,-102.710,450.254,174.794,15.777,152.423
C08903=1091.816,-102.960,450.264,174.793,15.777,152.423
C08904=1091.810,-103.210,450.273,174.791,15.776,152.423
C08905=1091.804,-103.459,450.284,174.789,15.775,152.423
C08906=1091.798,-103.709,450.294,174.788,15.775,152.424
C08907=1091.792,-103.959,450.303,174.786,15.775,152.424
C08908=1091.786,-104.208,450.313,174.785,15.773,152.424
C08909=1091.779,-104.458,450.323,174.783,15.773,152.424
C08910=1091.774,-104.708,450.333,174.782,15.773,152.424
C08911=1091.768,-104.958,450.343,174.780,15.772,152.425
C08912=1091.762,-105.207,450.352,174.778,15.771,152.425
C08913=1091.755,-105.457,450.362,174.777,15.771,152.425
C08914=1091.750,-105.707,450.373,174.775,15.770,152.425
C08915=1091.744,-105.956,450.382,174.773,15.769,152.426
C08916=1091.737,-106.206,450.392,174.772,15.769,152.426
C08917=1091.731,-106.456,450.402,174.770,15.769,152.426
C08918=1091.725,-106.706,450.411,174.769,15.768,152.426
C08919=1091.719,-106.955,450.422,174.768,15.768,152.426
C08920=1091.713,-107.205,450.432,174.766,15.767,152.427
C08921=1091.707,-107.455,450.441,174.764,15.766,152.427
C08922=1091.701,-107.705,450.451,174.762,15.766,152.427
C08923=1091.695,-107.955,450.460,174.761,15.765,152.427
C08924=1091.688,-108.204,450.470,174.759,15.765,152.428
C08925=1091.682,-108.454,450.479,174.757,15.764,152.428
C08926=1091.676,-108.703,450.490,174.756,15.764,152.428
C08927=1091.670,-108.953,450.500,174.754,15.763,152.428
C08928=1091.664,-109.203,450.509,174.752,15.762,152.429
C08929=1091.658,-109.453,450.519,174.751,15.762,152.429
C08930=1091.652,-109.703,450.529,174.749,15.762,152.429
C08931=1091.646,-109.953,450.538,174.747,15.761,152.429
C08932=1091.639,-110.202,450.548,174.746,15.761,152.430
C08933=1091.633,-110.452,450.557,174.744,15.760,152.430
C08934=1091.627,-110.702,450.567,174.742,15.760,152.430
C08935=1091.621,-110.951,450.577,174.742,15.759,152.430
C08936=1091.614,-111.201,450.587,174.740,15.758,152.430
C08937=1091.608,-111.451,450.596,174.739,15.758,152.431
C08938=1091.602,-111.701,450.606,174.737,15.758,152.431
C08939=1091.596,-111.950,450.615,174.735,15.757,152.431
C08940=1091.591,-112.200,450.626,174.734,15.757,152.431
C08941=1091.585,-112.450,450.635,174.732,15.756,152.432
C08942=1091.577,-112.718,450.645,174.730,15.756,152.432
C08943=1091.571,-112.986,450.655,174.728,15.755,152.432
C08944=1091.564,-113.254,450.666,174.727,15.755,152.432
C08945=1091.558,-113.521,450.676,174.725,15.754,152.433
C08946=1091.552,-113.771,450.685,174.723,15.754,152.433
C08947=1091.546,-114.021,450.695,174.722,15.754,152.433
C08948=1091.540,-114.271,450.704,174.720,15.753,152.433
C08949=1091.533,-114.521,450.714,174.718,15.752,152.434
C08950=1091.527,-114.770,450.724,174.717,15.752,152.434
C08951=1091.522,-115.020,450.733,174.715,15.752,152.434
C08952=1091.516,-115.269,450.742,174.713,15.751,152.435
C08953=1091.509,-115.519,450.752,174.712,15.751,152.435
C08954=1091.503,-115.769,450.761,174.710,15.750,152.435
C08955=1091.497,-116.019,450.771,174.708,15.750,152.435
C08956=1091.491,-116.268,450.781,174.708,15.749,152.435
C08957=1091.485,-116.518,450.790,174.706,15.748,152.436
C08958=1091.479,-116.768,450.800,174.705,15.748,152.436
C08959=1091.472,-117.018,450.809,174.703,15.748,152.436
C08960=1091.466,-117.268,450.819,174.701,15.747,152.436
C08961=1091.460,-117.517,450.828,174.700,15.747,152.437
C08962=1091.455,-117.767,450.837,174.698,15.746,152.437
C08963=1091.449,-118.017,450.846,174.697,15.746,152.437
C08964=1091.442,-118.267,450.856,174.694,15.746,152.437
C08965=1091.435,-118.516,450.865,174.693,15.745,152.438
C08966=1091.429,-118.766,450.875,174.691,15.745,152.438
C08967=1091.423,-119.016,450.884,174.690,15.745,152.438
C08968=1091.417,-119.266,450.894,174.688,15.744,152.439
C08969=1091.411,-119.515,450.903,174.687,15.744,152.439
C08970=1091.405,-119.765,450.913,174.685,15.743,152.439
C08971=1091.399,-120.014,450.922,174.684,15.743,152.439
C08972=1091.393,-120.265,450.931,174.682,15.743,152.439
C08973=1091.387,-120.515,450.940,174.680,15.742,152.440
C08974=1091.380,-120.764,450.949,174.679,15.742,152.440
C08975=1091.374,-121.014,450.959,174.677,15.741,152.440
C08976=1091.368,-121.264,450.969,174.676,15.741,152.440
C08977=1091.362,-121.513,450.978,174.674,15.740,152.441
C08978=1091.356,-121.763,450.987,174.672,15.740,152.441
C08979=1091.350,-122.013,450.996,174.671,15.740,152.441
C08980=1091.344,-122.263,451.006,174.669,15.739,152.442
C08981=1091.337,-122.512,451.015,174.668,15.739,152.442
C08982=1091.331,-122.762,451.024,174.666,15.738,152.442
C08983=1091.325,-123.012,451.034,174.664,15.738,152.442
C08984=1091.319,-123.262,451.042,174.662,15.738,152.443
C08985=1091.313,-123.511,451.052,174.661,15.738,152.443
C08986=1091.307,-123.761,451.062,174.659,15.737,152.443
C08987=1091.300,-124.011,451.070,174.658,15.737,152.443
C08988=1091.294,-124.260,451.080,174.656,15.737,152.444
C08989=1091.288,-124.511,451.089,174.655,15.736,152.444
C08990=1091.283,-124.760,451.098,174.653,15.735,152.444
C08991=1091.276,-125.010,451.108,174.651,15.735,152.444
C08992=1091.270,-125.259,451.117,174.650,15.735,152.445
C08993=1091.264,-125.510,451.125,174.648,15.735,152.445
C08994=1091.257,-125.759,451.135,174.646,15.735,152.445
C08995=1091.251,-126.009,451.145,174.645,15.734,152.446
C08996=1091.245,-126.258,451.153,174.643,15.734,152.446
C08997=1091.239,-126.508,451.162,174.641,15.733,152.446
C08998=1091.233,-126.758,451.172,174.640,15.733,152.446
C08999=1091.226,-127.008,451.181,174.638,15.732,152.447
C09000=1091.220,-127.258,451.190,174.637,15.733,152.447
C09001=1091.215,-127.507,451.199,174.635,15.732,152.447
C09002=1091.208,-127.767,451.208,174.634,15.732,152.447
C09003=1091.201,-128.025,451.218,174.632,15.732,152.448
C09004=1091.198,-128.285,451.228,174.630,15.730,152.448
C09005=1091.203,-128.541,451.241,174.630,15.727,152.447
C09006=1090.797,-128.563,451.122,174.587,15.834,152.477
C09007=1090.791,-128.306,451.109,174.587,15.837,152.477
C09008=1090.795,-128.047,451.099,174.589,15.838,152.477
C09009=1090.802,-127.788,451.089,174.591,15.839,152.477
C09010=1090.807,-127.529,451.079,174.592,15.839,152.476
C09011=1090.814,-127.280,451.070,174.594,15.839,152.476
C09012=1090.820,-127.030,451.062,174.596,15.840,152.476
C09013=1090.826,-126.780,451.052,174.597,15.840,152.476
C09014=1090.832,-126.531,451.043,174.599,15.841,152.475
C09015=1090.839,-126.281,451.034,174.600,15.841,152.475
C09016=1090.845,-126.031,451.025,174.602,15.841,152.475
C09017=1090.851,-125.781,451.015,174.603,15.841,152.475
C09018=1090.857,-125.531,451.006,174.605,15.842,152.474
C09019=1090.864,-125.281,450.998,174.607,15.842,152.474
C09020=1090.869,-125.032,450.988,174.608,15.842,152.474
C09021=1090.875,-124.782,450.979,174.610,15.843,152.474
C09022=1090.882,-124.532,450.969,174.611,15.843,152.473
C09023=1090.888,-124.282,450.961,174.613,15.844,152.473
C09024=1090.894,-124.032,450.951,174.615,15.844,152.473
C09025=1090.901,-123.783,450.942,174.616,15.844,152.473
C09026=1090.906,-123.534,450.933,174.618,15.845,152.472
C09027=1090.912,-123.284,450.923,174.619,15.845,152.472
C09028=1090.919,-123.034,450.915,174.621,15.846,152.472
C09029=1090.925,-122.784,450.905,174.623,15.846,152.472
C09030=1090.931,-122.534,450.896,174.624,15.846,152.471
C09031=1090.937,-122.284,450.886,174.626,15.847,152.471
C09032=1090.943,-122.035,450.877,174.627,15.847,152.471
C09033=1090.949,-121.785,450.868,174.629,15.848,152.471
C09034=1090.955,-121.535,450.858,174.631,15.848,152.470
C09035=1090.962,-121.285,450.849,174.632,15.848,152.470
C09036=1090.968,-121.036,450.840,174.634,15.848,152.470
C09037=1090.974,-120.786,450.830,174.635,15.849,152.469
C09038=1090.980,-120.537,450.821,174.637,15.849,152.469
C09039=1090.986,-120.287,450.812,174.639,15.850,152.469
C09040=1090.992,-120.037,450.803,174.640,15.850,152.469
C09041=1090.998,-119.787,450.793,174.642,15.851,152.468
C09042=1091.004,-119.537,450.784,174.643,15.851,152.468
C09043=1091.011,-119.287,450.775,174.645,15.851,152.468
C09044=1091.017,-119.038,450.765,174.647,15.852,152.468
C09045=1091.023,-118.788,450.755,174.648,15.852,152.468
C09046=1091.029,-118.539,450.746,174.650,15.853,152.467
C09047=1091.035,-118.289,450.737,174.651,15.853,152.467
C09048=1091.041,-118.039,450.727,174.653,15.854,152.467
C09049=1091.047,-117.789,450.718,174.655,15.854,152.467
C09050=1091.053,-117.539,450.709,174.656,15.855,152.466
C09051=1091.060,-117.289,450.699,174.658,15.855,152.466
C09052=1091.066,-117.039,450.690,174.660,15.856,152.466
C09053=1091.072,-116.790,450.680,174.661,15.856,152.466
C09054=1091.078,-116.540,450.670,174.663,15.857,152.465
C09055=1091.084,-116.291,450.661,174.665,15.857,152.465
C09056=1091.091,-116.041,450.652,174.666,15.857,152.465
C09057=1091.097,-115.791,450.643,174.668,15.858,152.465
C09058=1091.103,-115.542,450.633,174.669,15.858,152.464
C09059=1091.109,-115.292,450.624,174.671,15.859,152.464
C09060=1091.115,-115.042,450.614,174.672,15.859,152.464
C09061=1091.121,-114.792,450.604,174.674,15.859,152.464
C09062=1091.128,-114.542,450.595,174.676,15.860,152.463
C09063=1091.134,-114.293,450.585,174.677,15.861,152.463
C09064=1091.140,-114.043,450.576,174.678,15.861,152.463
C09065=1091.146,-113.793,450.566,174.680,15.862,152.463
C09066=1091.152,-113.543,450.557,174.682,15.862,152.462
C09067=1091.158,-113.275,450.547,174.683,15.862,152.462
C09068=1091.165,-113.007,450.536,174.685,15.863,152.462
C09069=1091.171,-112.739,450.526,174.687,15.864,152.462
C09070=1091.178,-112.470,450.516,174.689,15.864,152.461
C09071=1091.184,-112.221,450.506,174.690,15.864,152.461
C09072=1091.190,-111.971,450.497,174.692,15.865,152.461
C09073=1091.196,-111.721,450.486,174.694,15.866,152.461
C09074=1091.202,-111.471,450.477,174.695,15.866,152.461
C09075=1091.208,-111.221,450.467,174.696,15.867,152.460
C09076=1091.214,-110.971,450.458,174.698,15.868,152.460
C09077=1091.221,-110.722,450.447,174.699,15.868,152.460
C09078=1091.227,-110.472,450.438,174.701,15.868,152.460
C09079=1091.233,-110.223,450.428,174.703,15.869,152.459
C09080=1091.239,-109.973,450.419,174.704,15.869,152.459
C09081=1091.245,-109.724,450.410,174.706,15.870,152.459
C09082=1091.251,-109.474,450.400,174.708,15.871,152.459
